C07275=1071.215,48.448,-66.641,172.994,24.716,154.444
C07276=1071.221,48.697,-66.658,172.995,24.719,154.444
C07277=1071.227,48.947,-66.674,172.996,24.722,154.444
C07278=1071.233,49.196,-66.690,172.998,24.724,154.445
C07279=1071.239,49.446,-66.706,172.999,24.727,154.445
C07280=1071.244,49.695,-66.723,173.001,24.730,154.445
C07281=1071.250,49.945,-66.739,173.002,24.733,154.446
C07282=1071.256,50.194,-66.756,173.004,24.735,154.446
C07283=1071.262,50.443,-66.772,173.005,24.738,154.446
C07284=1071.268,50.693,-66.788,173.006,24.741,154.447
C07285=1071.273,50.942,-66.805,173.008,24.743,154.447
C07286=1071.279,51.192,-66.821,173.009,24.746,154.448
C07287=1071.285,51.441,-66.838,173.010,24.748,154.448
C07288=1071.291,51.690,-66.854,173.012,24.751,154.448
C07289=1071.297,51.940,-66.870,173.013,24.754,154.449
C07290=1071.302,52.189,-66.887,173.014,24.757,154.449
C07291=1071.308,52.439,-66.903,173.017,24.759,154.449
C07292=1071.314,52.688,-66.919,173.018,24.762,154.450
C07293=1071.320,52.937,-66.936,173.019,24.764,154.450
C07294=1071.326,53.186,-66.953,173.020,24.767,154.450
C07295=1071.332,53.436,-66.969,173.022,24.770,154.451
C07296=1071.337,53.685,-66.986,173.023,24.773,154.451
C07297=1071.344,53.935,-67.002,173.025,24.775,154.451
C07298=1071.349,54.185,-67.019,173.026,24.778,154.452
C07299=1071.355,54.434,-67.035,173.027,24.780,154.452
C07300=1071.361,54.683,-67.052,173.028,24.783,154.452
C07301=1071.367,54.932,-67.069,173.031,24.786,154.453
C07302=1071.373,55.182,-67.086,173.032,24.789,154.453
C07303=1071.379,55.431,-67.102,173.033,24.791,154.453
C07304=1071.384,55.681,-67.118,173.035,24.794,154.454
C07305=1071.391,55.929,-67.135,173.036,24.796,154.454
C07306=1071.396,56.179,-67.152,173.037,24.799,154.454
C07307=1071.403,56.429,-67.169,173.039,24.802,154.455
C07308=1071.408,56.678,-67.185,173.040,24.805,154.455
C07309=1071.415,56.927,-67.202,173.041,24.807,154.455
C07310=1071.420,57.177,-67.219,173.043,24.810,154.456
C07311=1071.426,57.426,-67.235,173.045,24.812,154.456
C07312=1071.432,57.675,-67.251,173.046,24.815,154.456
C07313=1071.437,57.924,-67.269,173.048,24.818,154.457
C07314=1071.444,58.175,-67.285,173.049,24.821,154.457
C07315=1071.450,58.424,-67.302,173.050,24.823,154.457
C07316=1071.456,58.673,-67.318,173.052,24.826,154.458
C07317=1071.461,58.922,-67.335,173.053,24.828,154.458
C07318=1071.467,59.172,-67.352,173.054,24.831,154.458
C07319=1071.473,59.421,-67.368,173.056,24.833,154.459
C07320=1071.479,59.671,-67.386,173.057,24.836,154.459
C07321=1071.485,59.920,-67.402,173.059,24.839,154.459
C07322=1071.491,60.169,-67.418,173.061,24.841,154.460
C07323=1071.497,60.418,-67.436,173.062,24.844,154.460
C07324=1071.503,60.668,-67.452,173.063,24.847,154.460
C07325=1071.510,60.917,-67.470,173.065,24.850,154.461
C07326=1071.516,61.167,-67.486,173.066,24.852,154.461
C07327=1071.521,61.416,-67.503,173.067,24.855,154.461
C07328=1071.527,61.665,-67.520,173.069,24.857,154.462
C07329=1071.533,61.914,-67.536,173.070,24.860,154.462
C07330=1071.539,62.165,-67.553,173.072,24.863,154.462
C07331=1071.546,62.447,-67.572,173.073,24.866,154.463
C07332=1071.553,62.729,-67.592,173.075,24.869,154.463
C07333=1071.559,63.011,-67.610,173.077,24.872,154.464
C07334=1071.565,63.293,-67.630,173.078,24.875,154.464
C07335=1071.572,63.543,-67.646,173.080,24.877,154.464
C07336=1071.578,63.792,-67.663,173.081,24.879,154.465
C07337=1071.583,64.041,-67.680,173.082,24.882,154.465
C07338=1071.590,64.291,-67.697,173.085,24.885,154.465
C07339=1071.596,64.540,-67.714,173.086,24.888,154.466
C07340=1071.602,64.789,-67.731,173.087,24.890,154.466
C07341=1071.607,65.039,-67.748,173.089,24.893,154.466
C07342=1071.613,65.287,-67.765,173.090,24.895,154.467
C07343=1071.619,65.538,-67.782,173.091,24.898,154.467
C07344=1071.625,65.787,-67.799,173.093,24.901,154.467
C07345=1071.631,66.036,-67.816,173.094,24.904,154.468
C07346=1071.637,66.285,-67.833,173.096,24.906,154.468
C07347=1071.643,66.535,-67.851,173.097,24.909,154.468
C07348=1071.648,66.784,-67.868,173.099,24.911,154.469
C07349=1071.654,67.033,-67.885,173.100,24.914,154.469
C07350=1071.660,67.283,-67.902,173.102,24.917,154.469
C07351=1071.666,67.532,-67.919,173.103,24.920,154.470
C07352=1071.672,67.781,-67.936,173.104,24.922,154.470
C07353=1071.678,68.031,-67.953,173.106,24.925,154.470
C07354=1071.683,68.280,-67.970,173.107,24.927,154.471
C07355=1071.689,68.530,-67.988,173.109,24.930,154.471
C07356=1071.696,68.779,-68.005,173.111,24.933,154.471
C07357=1071.701,69.028,-68.022,173.112,24.936,154.472
C07358=1071.706,69.277,-68.039,173.113,24.939,154.472
C07359=1071.713,69.527,-68.056,173.114,24.941,154.472
C07360=1071.719,69.776,-68.074,173.116,24.944,154.473
C07361=1071.724,70.026,-68.091,173.117,24.946,154.473
C07362=1071.731,70.275,-68.108,173.118,24.949,154.473
C07363=1071.736,70.524,-68.126,173.121,24.952,154.474
C07364=1071.741,70.774,-68.142,173.122,24.955,154.474
C07365=1071.748,71.022,-68.159,173.123,24.957,154.474
C07366=1071.754,71.272,-68.177,173.125,24.960,154.475
C07367=1071.759,71.522,-68.194,173.126,24.962,154.475
C07368=1071.765,71.771,-68.212,173.127,24.965,154.476
C07369=1071.771,72.020,-68.229,173.129,24.967,154.476
C07370=1071.777,72.269,-68.247,173.131,24.971,154.476
C07371=1071.782,72.519,-68.264,173.132,24.973,154.476
C07372=1071.788,72.769,-68.281,173.134,24.976,154.477
C07373=1071.794,73.017,-68.298,173.135,24.979,154.477
C07374=1071.800,73.266,-68.316,173.136,24.981,154.478
C07375=1071.806,73.516,-68.334,173.138,24.984,154.478
C07376=1071.811,73.766,-68.351,173.139,24.986,154.478
C07377=1071.817,74.015,-68.368,173.140,24.989,154.479
C07378=1071.823,74.264,-68.385,173.143,24.992,154.479
C07379=1071.829,74.513,-68.403,173.144,24.995,154.479
C07380=1071.835,74.762,-68.421,173.145,24.997,154.480
C07381=1071.841,75.012,-68.439,173.147,25.000,154.480
C07382=1071.846,75.262,-68.456,173.148,25.002,154.480
C07383=1071.852,75.511,-68.473,173.149,25.005,154.481
C07384=1071.858,75.760,-68.490,173.151,25.008,154.481
C07385=1071.864,76.009,-68.508,173.153,25.011,154.481
C07386=1071.870,76.258,-68.526,173.154,25.013,154.482
C07387=1071.876,76.508,-68.544,173.156,25.016,154.482
C07388=1071.882,76.757,-68.561,173.157,25.018,154.482
C07389=1071.887,77.006,-68.578,173.158,25.021,154.483
C07390=1071.893,77.256,-68.595,173.160,25.024,154.483
C07391=1071.899,77.505,-68.613,173.161,25.026,154.483
C07392=1071.905,77.755,-68.631,173.163,25.029,154.484
C07393=1071.910,78.004,-68.648,173.165,25.032,154.484
C07394=1071.916,78.253,-68.666,173.166,25.034,154.484
C07395=1071.923,78.536,-68.686,173.167,25.037,154.485
C07396=1071.930,78.818,-68.706,173.170,25.040,154.485
C07397=1071.936,79.100,-68.726,173.171,25.043,154.486
C07398=1071.943,79.382,-68.746,173.172,25.046,154.486
C07399=1071.948,79.631,-68.763,173.174,25.049,154.486
C07400=1071.954,79.880,-68.781,173.176,25.052,154.487
C07401=1071.960,80.130,-68.799,173.177,25.055,154.487
C07402=1071.966,80.379,-68.816,173.178,25.058,154.487
C07403=1071.972,80.629,-68.834,173.180,25.060,154.488
C07404=1071.977,80.878,-68.852,173.181,25.063,154.488
C07405=1071.983,81.127,-68.869,173.183,25.065,154.488
C07406=1071.989,81.377,-68.887,173.185,25.068,154.489
C07407=1071.995,81.625,-68.906,173.186,25.071,154.489
C07408=1072.001,81.875,-68.924,173.187,25.074,154.489
C07409=1072.006,82.124,-68.941,173.189,25.076,154.490
C07410=1072.012,82.373,-68.959,173.190,25.079,154.490
C07411=1072.018,82.622,-68.977,173.191,25.082,154.491
C07412=1072.023,82.872,-68.995,173.194,25.084,154.491
C07413=1072.029,83.122,-69.013,173.195,25.087,154.491
C07414=1072.034,83.371,-69.030,173.196,25.090,154.491
C07415=1072.040,83.620,-69.048,173.198,25.092,154.492
C07416=1072.046,83.869,-69.066,173.199,25.095,154.492
C07417=1072.052,84.119,-69.085,173.200,25.098,154.493
C07418=1072.058,84.368,-69.102,173.203,25.100,154.493
C07419=1072.063,84.617,-69.120,173.204,25.103,154.493
C07420=1072.070,84.866,-69.138,173.205,25.105,154.494
C07421=1072.075,85.115,-69.155,173.207,25.108,154.494
C07422=1072.081,85.365,-69.173,173.208,25.111,154.494
C07423=1072.087,85.614,-69.191,173.209,25.114,154.495
C07424=1072.093,85.863,-69.209,173.212,25.116,154.495
C07425=1072.099,86.112,-69.227,173.213,25.119,154.495
C07426=1072.104,86.362,-69.245,173.215,25.121,154.496
C07427=1072.110,86.611,-69.263,173.216,25.124,154.496
C07428=1072.116,86.861,-69.282,173.217,25.127,154.496
C07429=1072.122,87.110,-69.299,173.219,25.130,154.497
C07430=1072.128,87.359,-69.317,173.221,25.132,154.497
C07431=1072.133,87.608,-69.335,173.222,25.135,154.497
C07432=1072.140,87.857,-69.353,173.224,25.137,154.498
C07433=1072.146,88.107,-69.371,173.225,25.140,154.498
C07434=1072.151,88.356,-69.389,173.226,25.143,154.498
C07435=1072.157,88.606,-69.408,173.228,25.146,154.499
C07436=1072.162,88.855,-69.426,173.230,25.148,154.499
C07437=1072.169,89.104,-69.444,173.231,25.150,154.499
C07438=1072.174,89.353,-69.462,173.233,25.153,154.500
C07439=1072.181,89.603,-69.480,173.234,25.156,154.500
C07440=1072.186,89.852,-69.497,173.235,25.159,154.500
C07441=1072.192,90.101,-69.516,173.237,25.161,154.501
C07442=1072.199,90.351,-69.534,173.239,25.164,154.501
C07443=1072.203,90.600,-69.552,173.240,25.166,154.501
C07444=1072.210,90.849,-69.571,173.242,25.169,154.502
C07445=1072.215,91.098,-69.588,173.243,25.172,154.502
C07446=1072.221,91.348,-69.606,173.244,25.175,154.502
C07447=1072.226,91.597,-69.625,173.246,25.177,154.503
C07448=1072.233,91.846,-69.643,173.248,25.180,154.503
C07449=1072.238,92.095,-69.661,173.250,25.182,154.503
C07450=1072.244,92.345,-69.680,173.251,25.185,154.504
C07451=1072.250,92.595,-69.698,173.252,25.188,154.504
C07452=1072.255,92.843,-69.717,173.254,25.190,154.504
C07453=1072.261,93.093,-69.735,173.256,25.193,154.505
C07454=1072.267,93.341,-69.753,173.257,25.196,154.505
C07455=1072.272,93.591,-69.771,173.259,25.198,154.505
C07456=1072.278,93.840,-69.790,173.260,25.201,154.506
C07457=1072.284,94.090,-69.808,173.261,25.204,154.506
C07458=1072.290,94.339,-69.827,173.264,25.207,154.506
C07459=1072.297,94.621,-69.847,173.265,25.210,154.507
C07460=1072.303,94.903,-69.868,173.266,25.212,154.507
C07461=1072.309,95.186,-69.889,173.268,25.216,154.508
C07462=1072.316,95.467,-69.909,173.270,25.219,154.508
C07463=1072.322,95.717,-69.929,173.272,25.221,154.508
C07464=1072.327,95.966,-69.946,173.273,25.224,154.509
C07465=1072.334,96.215,-69.965,173.275,25.226,154.509
C07466=1072.339,96.464,-69.983,173.276,25.229,154.509
C07467=1072.345,96.713,-70.002,173.277,25.232,154.510
C07468=1072.350,96.964,-70.020,173.280,25.235,154.510
C07469=1072.356,97.212,-70.038,173.281,25.237,154.510
C07470=1072.363,97.461,-70.057,173.282,25.240,154.511
C07471=1072.368,97.711,-70.076,173.284,25.242,154.511
C07472=1072.374,97.960,-70.094,173.285,25.245,154.511
C07473=1072.379,98.210,-70.112,173.288,25.248,154.512
C07474=1072.386,98.459,-70.131,173.289,25.251,154.512
C07475=1072.391,98.707,-70.150,173.290,25.253,154.512
C07476=1072.397,98.957,-70.168,173.292,25.255,154.513
C07477=1072.403,99.206,-70.186,173.293,25.258,154.513
C07478=1072.408,99.455,-70.205,173.295,25.261,154.513
C07479=1072.414,99.705,-70.223,173.297,25.264,154.514
C07480=1072.420,99.954,-70.243,173.298,25.266,154.514
C07481=1072.427,100.203,-70.261,173.299,25.269,154.514
C07482=1072.431,100.453,-70.279,173.301,25.271,154.515
C07483=1072.438,100.702,-70.298,173.303,25.274,154.515
C07484=1072.444,100.951,-70.317,173.304,25.277,154.515
C07485=1072.449,101.200,-70.336,173.306,25.279,154.516
C07486=1072.455,101.450,-70.354,173.307,25.282,154.516
C07487=1072.461,101.699,-70.373,173.310,25.285,154.516
C07488=1072.466,101.948,-70.392,173.311,25.287,154.517
C07489=1072.473,102.197,-70.410,173.312,25.290,154.517
C07490=1072.478,102.447,-70.429,173.314,25.293,154.517
C07491=1072.483,102.695,-70.448,173.315,25.295,154.518
C07492=1072.489,102.945,-70.466,173.317,25.298,154.518
C07493=1072.495,103.194,-70.486,173.319,25.300,154.518
C07494=1072.500,103.443,-70.504,173.320,25.303,154.519
C07495=1072.506,103.693,-70.522,173.321,25.306,154.519
C07496=1072.512,103.942,-70.542,173.323,25.309,154.519
C07497=1072.518,104.191,-70.561,173.325,25.311,154.520
C07498=1072.524,104.440,-70.579,173.326,25.314,154.520
C07499=1072.529,104.689,-70.598,173.328,25.316,154.520
C07500=1072.535,104.939,-70.618,173.329,25.319,154.521
C07501=1072.541,105.187,-70.636,173.332,25.322,154.521
C07502=1072.546,105.437,-70.654,173.333,25.325,154.522
C07503=1072.552,105.687,-70.674,173.334,25.327,154.522
C07504=1072.558,105.936,-70.692,173.336,25.330,154.522
C07505=1072.563,106.184,-70.711,173.338,25.333,154.522
C07506=1072.569,106.434,-70.730,173.339,25.335,154.523
C07507=1072.575,106.683,-70.749,173.341,25.338,154.523
C07508=1072.581,106.932,-70.768,173.342,25.341,154.524
C07509=1072.586,107.181,-70.787,173.343,25.343,154.524
C07510=1072.593,107.430,-70.806,173.346,25.346,154.524
C07511=1072.598,107.680,-70.825,173.347,25.348,154.525
C07512=1072.604,107.929,-70.844,173.349,25.351,154.525
C07513=1072.610,108.178,-70.863,173.350,25.354,154.525
C07514=1072.616,108.427,-70.882,173.352,25.356,154.525
C07515=1072.621,108.676,-70.901,173.354,25.359,154.526
C07516=1072.627,108.926,-70.920,173.355,25.361,154.526
C07517=1072.633,109.175,-70.939,173.356,25.364,154.527
C07518=1072.639,109.424,-70.958,173.359,25.367,154.527
C07519=1072.644,109.673,-70.977,173.360,25.369,154.527
C07520=1072.651,109.922,-70.996,173.361,25.372,154.528
C07521=1072.656,110.172,-71.015,173.363,25.374,154.528
C07522=1072.662,110.421,-71.034,173.365,25.378,154.528
C07523=1072.669,110.704,-71.056,173.367,25.380,154.528
C07524=1072.675,110.985,-71.077,173.369,25.383,154.529
C07525=1072.682,111.268,-71.099,173.370,25.386,154.529
C07526=1072.688,111.550,-71.120,173.372,25.389,154.530
C07527=1072.694,111.800,-71.139,173.374,25.391,154.530
C07528=1072.700,112.049,-71.159,173.375,25.394,154.530
C07529=1072.705,112.297,-71.178,173.377,25.397,154.531
C07530=1072.711,112.547,-71.197,173.379,25.400,154.531
C07531=1072.717,112.796,-71.217,173.380,25.402,154.531
C07532=1072.722,113.046,-71.236,173.382,25.405,154.532
C07533=1072.729,113.295,-71.254,173.384,25.408,154.532
C07534=1072.734,113.544,-71.274,173.385,25.410,154.532
C07535=1072.740,113.793,-71.294,173.387,25.413,154.533
C07536=1072.745,114.042,-71.313,173.388,25.415,154.533
C07537=1072.751,114.291,-71.332,173.390,25.418,154.533
C07538=1072.757,114.541,-71.351,173.392,25.421,154.534
C07539=1072.763,114.790,-71.370,173.393,25.423,154.534
C07540=1072.768,115.039,-71.390,173.395,25.426,154.534
C07541=1072.774,115.288,-71.410,173.397,25.429,154.535
C07542=1072.779,115.537,-71.428,173.398,25.431,154.535
C07543=1072.785,115.786,-71.448,173.400,25.434,154.535
C07544=1072.791,116.035,-71.468,173.401,25.437,154.536
C07545=1072.797,116.285,-71.487,173.403,25.440,154.536
C07546=1072.802,116.534,-71.506,173.405,25.442,154.536
C07547=1072.807,116.784,-71.526,173.406,25.445,154.537
C07548=1072.813,117.032,-71.546,173.408,25.448,154.537
C07549=1072.818,117.281,-71.565,173.410,25.450,154.537
C07550=1072.824,117.531,-71.584,173.411,25.453,154.538
C07551=1072.830,117.780,-71.604,173.412,25.455,154.538
C07552=1072.836,118.029,-71.623,173.415,25.458,154.538
C07553=1072.841,118.278,-71.642,173.416,25.461,154.539
C07554=1072.847,118.527,-71.662,173.418,25.463,154.539
C07555=1072.853,118.777,-71.682,173.419,25.466,154.539
C07556=1072.858,119.025,-71.701,173.421,25.469,154.540
C07557=1072.863,119.275,-71.721,173.423,25.471,154.540
C07558=1072.869,119.524,-71.740,173.424,25.474,154.540
C07559=1072.875,119.773,-71.760,173.426,25.477,154.541
C07560=1072.881,120.022,-71.780,173.428,25.479,154.541
C07561=1072.886,120.272,-71.799,173.429,25.482,154.541
C07562=1072.892,120.520,-71.819,173.431,25.484,154.542
C07563=1072.898,120.770,-71.838,173.433,25.488,154.542
C07564=1072.904,121.019,-71.858,173.434,25.490,154.542
C07565=1072.909,121.268,-71.878,173.436,25.492,154.543
C07566=1072.915,121.518,-71.897,173.438,25.495,154.543
C07567=1072.921,121.767,-71.917,173.439,25.498,154.543
C07568=1072.926,122.016,-71.936,173.441,25.501,154.544
C07569=1072.932,122.265,-71.956,173.443,25.503,154.544
C07570=1072.938,122.514,-71.975,173.444,25.506,154.544
C07571=1072.944,122.763,-71.995,173.446,25.508,154.545
C07572=1072.949,123.013,-72.015,173.447,25.511,154.545
C07573=1072.955,123.262,-72.035,173.450,25.514,154.545
C07574=1072.961,123.511,-72.054,173.451,25.516,154.546
C07575=1072.967,123.760,-72.074,173.452,25.519,154.546
C07576=1072.972,124.009,-72.094,173.455,25.522,154.546
C07577=1072.978,124.258,-72.114,173.456,25.524,154.547
C07578=1072.984,124.507,-72.134,173.458,25.527,154.547
C07579=1072.989,124.757,-72.153,173.460,25.529,154.547
C07580=1072.995,125.006,-72.173,173.461,25.532,154.548
C07581=1073.001,125.255,-72.193,173.463,25.535,154.548
C07582=1073.007,125.504,-72.213,173.465,25.537,154.548
C07583=1073.012,125.754,-72.232,173.466,25.540,154.549
C07584=1073.018,126.002,-72.252,173.468,25.542,154.549
C07585=1073.024,126.251,-72.272,173.469,25.545,154.549
C07586=1073.030,126.501,-72.292,173.472,25.548,154.550
C07587=1073.036,126.783,-72.314,173.473,25.551,154.550
C07588=1073.043,127.065,-72.336,173.475,25.553,154.550
C07589=1073.049,127.347,-72.359,173.478,25.556,154.551
C07590=1073.055,127.630,-72.382,173.479,25.559,154.551
C07591=1073.061,127.878,-72.402,173.481,25.562,154.551
C07592=1073.067,128.127,-72.422,173.483,25.565,154.552
C07593=1073.073,128.376,-72.442,173.484,25.567,154.552
C07594=1073.078,128.626,-72.461,173.486,25.570,154.552
C07595=1073.084,128.875,-72.481,173.488,25.572,154.553
C07596=1073.090,129.123,-72.501,173.489,25.575,154.553
C07597=1073.097,129.374,-72.521,173.492,25.577,154.553
C07598=1073.102,129.623,-72.541,173.493,25.580,154.554
C07599=1073.108,129.871,-72.561,173.494,25.583,154.554
C07600=1073.114,130.120,-72.581,173.497,25.585,154.554
C07601=1073.120,130.370,-72.601,173.498,25.588,154.555
C07602=1073.125,130.619,-72.621,173.500,25.590,154.555
C07603=1073.131,130.868,-72.641,173.502,25.593,154.555
C07604=1073.137,131.117,-72.661,173.503,25.595,154.555
C07605=1073.143,131.366,-72.681,173.505,25.598,154.556
C07606=1073.148,131.616,-72.701,173.507,25.601,154.556
C07607=1073.154,131.865,-72.721,173.509,25.603,154.556
C07608=1073.160,132.113,-72.741,173.510,25.606,154.557
C07609=1073.166,132.362,-72.762,173.512,25.608,154.557
C07610=1073.172,132.611,-72.782,173.514,25.611,154.557
C07611=1073.177,132.860,-72.802,173.515,25.614,154.558
C07612=1073.183,133.111,-72.822,173.517,25.616,154.558
C07613=1073.188,133.360,-72.842,173.519,25.619,154.558
C07614=1073.194,133.608,-72.862,173.521,25.622,154.559
C07615=1073.200,133.858,-72.883,173.523,25.625,154.559
C07616=1073.206,134.106,-72.903,173.524,25.627,154.559
C07617=1073.211,134.356,-72.923,173.526,25.629,154.560
C07618=1073.217,134.604,-72.943,173.528,25.632,154.560
C07619=1073.223,134.854,-72.964,173.529,25.635,154.560
C07620=1073.229,135.103,-72.984,173.532,25.637,154.561
C07621=1073.234,135.352,-73.005,173.533,25.640,154.561
C07622=1073.240,135.601,-73.025,173.534,25.642,154.561
C07623=1073.245,135.850,-73.045,173.537,25.645,154.562
C07624=1073.251,136.099,-73.065,173.538,25.648,154.562
C07625=1073.257,136.349,-73.086,173.540,25.650,154.562
C07626=1073.263,136.597,-73.106,173.542,25.653,154.563
C07627=1073.268,136.847,-73.127,173.543,25.655,154.563
C07628=1073.274,137.095,-73.147,173.546,25.658,154.563
C07629=1073.280,137.345,-73.167,173.547,25.661,154.564
C07630=1073.286,137.593,-73.187,173.548,25.663,154.564
C07631=1073.292,137.843,-73.208,173.551,25.666,154.564
C07632=1073.297,138.092,-73.229,173.552,25.669,154.564
C07633=1073.303,138.341,-73.249,173.555,25.671,154.565
C07634=1073.308,138.590,-73.269,173.556,25.674,154.565
C07635=1073.315,138.840,-73.289,173.557,25.676,154.565
C07636=1073.320,139.089,-73.310,173.560,25.679,154.566
C07637=1073.325,139.338,-73.331,173.561,25.682,154.566
C07638=1073.331,139.587,-73.351,173.563,25.684,154.566
C07639=1073.337,139.835,-73.372,173.565,25.687,154.567
C07640=1073.343,140.085,-73.392,173.566,25.690,154.567
C07641=1073.349,140.334,-73.413,173.569,25.692,154.567
C07642=1073.354,140.583,-73.433,173.570,25.695,154.568
C07643=1073.360,140.832,-73.453,173.572,25.697,154.568
C07644=1073.366,141.082,-73.474,173.574,25.700,154.568
C07645=1073.371,141.330,-73.495,173.575,25.703,154.569
C07646=1073.376,141.579,-73.516,173.578,25.705,154.569
C07647=1073.382,141.828,-73.536,173.579,25.708,154.569
C07648=1073.388,142.078,-73.557,173.580,25.711,154.570
C07649=1073.394,142.327,-73.577,173.583,25.713,154.570
C07650=1073.399,142.576,-73.599,173.584,25.715,154.570
C07651=1073.405,142.858,-73.621,173.587,25.719,154.571
C07652=1073.412,143.140,-73.645,173.589,25.722,154.571
C07653=1073.419,143.422,-73.668,173.590,25.725,154.571
C07654=1073.425,143.704,-73.692,173.592,25.728,154.572
C07655=1073.431,143.953,-73.712,173.595,25.730,154.572
C07656=1073.436,144.202,-73.733,173.596,25.733,154.572
C07657=1073.442,144.451,-73.755,173.598,25.735,154.573
C07658=1073.448,144.700,-73.775,173.600,25.738,154.573
C07659=1073.453,144.949,-73.796,173.602,25.740,154.573
C07660=1073.460,145.198,-73.817,173.604,25.743,154.574
C07661=1073.465,145.447,-73.837,173.605,25.746,154.574
C07662=1073.470,145.697,-73.858,173.608,25.748,154.574
C07663=1073.476,145.945,-73.879,173.609,25.751,154.575
C07664=1073.482,146.195,-73.900,173.611,25.753,154.575
C07665=1073.488,146.444,-73.920,173.613,25.756,154.575
C07666=1073.493,146.692,-73.941,173.614,25.759,154.576
C07667=1073.499,146.942,-73.962,173.617,25.762,154.576
C07668=1073.505,147.191,-73.983,173.618,25.764,154.576
C07669=1073.511,147.440,-74.004,173.620,25.767,154.576
C07670=1073.517,147.689,-74.024,173.622,25.769,154.577
C07671=1073.522,147.938,-74.046,173.623,25.772,154.577
C07672=1073.528,148.188,-74.067,173.626,25.775,154.577
C07673=1073.533,148.436,-74.088,173.627,25.777,154.578
C07674=1073.539,148.685,-74.108,173.630,25.780,154.578
C07675=1073.545,148.934,-74.130,173.631,25.782,154.578
C07676=1073.550,149.183,-74.151,173.633,25.785,154.579
C07677=1073.556,149.432,-74.172,173.635,25.788,154.579
C07678=1073.562,149.682,-74.193,173.637,25.790,154.579
C07679=1073.567,149.930,-74.214,173.638,25.793,154.580
C07680=1073.572,150.179,-74.235,173.640,25.796,154.580
C07681=1073.579,150.429,-74.256,173.642,25.798,154.580
C07682=1073.584,150.678,-74.277,173.644,25.800,154.581
C07683=1073.590,150.927,-74.298,173.646,25.804,154.581
C07684=1073.595,151.176,-74.319,173.647,25.806,154.581
C07685=1073.601,151.425,-74.340,173.650,25.808,154.581
C07686=1073.607,151.674,-74.362,173.651,25.811,154.582
C07687=1073.612,151.923,-74.382,173.654,25.814,154.582
C07688=1073.618,152.172,-74.404,173.655,25.817,154.583
C07689=1073.624,152.421,-74.425,173.657,25.819,154.583
C07690=1073.629,152.670,-74.446,173.659,25.822,154.583
C07691=1073.635,152.919,-74.467,173.660,25.824,154.584
C07692=1073.641,153.168,-74.488,173.663,25.827,154.584
C07693=1073.647,153.417,-74.510,173.664,25.829,154.584
C07694=1073.652,153.666,-74.531,173.666,25.832,154.584
C07695=1073.658,153.915,-74.551,173.668,25.835,154.585
C07696=1073.664,154.164,-74.573,173.670,25.837,154.585
C07697=1073.669,154.413,-74.594,173.672,25.840,154.585
C07698=1073.675,154.662,-74.615,173.674,25.843,154.586
C07699=1073.681,154.911,-74.637,173.676,25.845,154.586
C07700=1073.687,155.160,-74.658,173.678,25.848,154.586
C07701=1073.691,155.410,-74.679,173.679,25.850,154.587
C07702=1073.698,155.659,-74.701,173.682,25.853,154.587
C07703=1073.703,155.907,-74.722,173.683,25.856,154.587
C07704=1073.709,156.156,-74.744,173.685,25.858,154.588
C07705=1073.715,156.406,-74.764,173.687,25.861,154.588
C07706=1073.720,156.654,-74.786,173.689,25.864,154.588
C07707=1073.726,156.904,-74.808,173.691,25.866,154.588
C07708=1073.731,157.152,-74.829,173.693,25.869,154.589
C07709=1073.737,157.401,-74.851,173.694,25.872,154.589
C07710=1073.743,157.650,-74.871,173.697,25.874,154.589
C07711=1073.749,157.900,-74.893,173.698,25.877,154.590
C07712=1073.754,158.148,-74.914,173.701,25.880,154.590
C07713=1073.760,158.398,-74.937,173.702,25.882,154.590
C07714=1073.765,158.646,-74.958,173.704,25.885,154.591
C07715=1073.772,158.929,-74.982,173.707,25.888,154.591
C07716=1073.779,159.210,-75.006,173.708,25.890,154.591
C07717=1073.784,159.492,-75.030,173.710,25.893,154.592
C07718=1073.791,159.774,-75.055,173.713,25.897,154.592
C07719=1073.797,160.023,-75.077,173.715,25.899,154.592
C07720=1073.803,160.272,-75.098,173.717,25.901,154.593
C07721=1073.808,160.520,-75.120,173.719,25.905,154.593
C07722=1073.814,160.770,-75.142,173.720,25.907,154.593
C07723=1073.819,161.018,-75.163,173.723,25.909,154.594
C07724=1073.826,161.267,-75.185,173.724,25.912,154.594
C07725=1073.832,161.517,-75.206,173.727,25.915,154.594
C07726=1073.837,161.766,-75.228,173.728,25.918,154.595
C07727=1073.841,162.014,-75.250,173.730,25.920,154.595
C07728=1073.848,162.264,-75.272,173.732,25.923,154.595
C07729=1073.852,162.512,-75.294,173.734,25.926,154.596
C07730=1073.858,162.762,-75.315,173.736,25.928,154.596
C07731=1073.866,163.133,-75.347,173.739,25.933,154.597
C07732=1073.874,163.505,-75.381,173.742,25.937,154.597
C07733=1073.883,163.877,-75.412,173.745,25.941,154.597
C07734=1073.891,164.249,-75.445,173.747,25.944,154.598
C07735=1073.896,164.498,-75.467,173.749,25.947,154.598
C07736=1073.902,164.747,-75.489,173.752,25.950,154.599
C07737=1073.907,164.996,-75.511,173.753,25.953,154.599
C07738=1073.913,165.245,-75.532,173.755,25.955,154.599
C07739=1073.918,165.494,-75.554,173.757,25.958,154.600
C07740=1073.924,165.742,-75.577,173.759,25.961,154.600
C07741=1073.930,165.992,-75.599,173.761,25.963,154.600
C07742=1073.935,166.240,-75.620,173.763,25.966,154.601
C07743=1073.941,166.490,-75.642,173.764,25.968,154.601
C07744=1073.946,166.739,-75.664,173.767,25.972,154.601
C07745=1073.952,166.987,-75.687,173.769,25.974,154.602
C07746=1073.957,167.236,-75.708,173.771,25.977,154.602
C07747=1073.963,167.485,-75.730,173.773,25.979,154.602
C07748=1073.969,167.735,-75.752,173.774,25.982,154.603
C07749=1073.973,167.984,-75.774,173.777,25.985,154.603
C07750=1073.980,168.232,-75.797,173.778,25.987,154.603
C07751=1073.985,168.481,-75.818,173.781,25.990,154.604
C07752=1073.991,168.730,-75.840,173.782,25.993,154.604
C07753=1073.996,168.980,-75.862,173.784,25.996,154.604
C07754=1074.001,169.228,-75.885,173.787,25.998,154.605
C07755=1074.008,169.477,-75.907,173.788,26.001,154.605
C07756=1074.013,169.727,-75.929,173.791,26.004,154.605
C07757=1074.019,169.975,-75.951,173.792,26.006,154.606
C07758=1074.024,170.224,-75.973,173.794,26.009,154.606
C07759=1074.030,170.474,-75.995,173.797,26.012,154.606
C07760=1074.036,170.721,-76.017,173.798,26.014,154.607
C07761=1074.041,170.971,-76.039,173.801,26.017,154.607
C07762=1074.046,171.221,-76.062,173.802,26.019,154.607
C07763=1074.052,171.468,-76.084,173.804,26.022,154.608
C07764=1074.058,171.718,-76.106,173.807,26.025,154.608
C07765=1074.063,171.967,-76.129,173.808,26.027,154.608
C07766=1074.069,172.215,-76.150,173.811,26.030,154.608
C07767=1074.074,172.465,-76.172,173.812,26.033,154.609
C07768=1074.080,172.714,-76.195,173.814,26.036,154.609
C07769=1074.086,172.963,-76.217,173.817,26.038,154.609
C07770=1074.091,173.211,-76.239,173.818,26.041,154.610
C07771=1074.097,173.461,-76.262,173.821,26.044,154.610
C07772=1074.103,173.709,-76.284,173.822,26.046,154.610
C07773=1074.109,173.959,-76.306,173.824,26.049,154.611
C07774=1074.114,174.207,-76.329,173.827,26.052,154.611
C07775=1074.123,174.614,-76.365,173.830,26.056,154.611
C07776=1074.132,175.022,-76.401,173.833,26.060,154.612
C07777=1074.142,175.430,-76.437,173.837,26.064,154.612
C07778=1074.152,175.838,-76.475,173.840,26.069,154.613
C07779=1074.156,176.087,-76.497,173.841,26.071,154.613
C07780=1074.163,176.335,-76.519,173.844,26.074,154.614
C07781=1074.169,176.584,-76.542,173.846,26.077,154.614
C07782=1074.174,176.834,-76.565,173.848,26.079,154.614
C07783=1074.180,177.082,-76.587,173.850,26.082,154.615
C07784=1074.185,177.331,-76.609,173.852,26.085,154.615
C07785=1074.191,177.580,-76.632,173.854,26.087,154.615
C07786=1074.197,177.829,-76.655,173.856,26.090,154.616
C07787=1074.203,178.078,-76.676,173.859,26.093,154.616
C07788=1074.209,178.327,-76.699,173.860,26.095,154.616
C07789=1074.215,178.576,-76.722,173.863,26.098,154.616
C07790=1074.220,178.825,-76.744,173.865,26.101,154.617
C07791=1074.226,179.073,-76.766,173.866,26.103,154.617
C07792=1074.232,179.322,-76.789,173.869,26.106,154.617
C07793=1074.237,179.572,-76.812,173.871,26.109,154.618
C07794=1074.243,179.820,-76.835,173.873,26.111,154.618
C07795=1074.249,180.069,-76.857,173.875,26.114,154.618
C07796=1074.255,180.318,-76.880,173.877,26.117,154.619
C07797=1074.260,180.567,-76.902,173.879,26.119,154.619
C07798=1074.266,180.816,-76.925,173.881,26.121,154.619
C07799=1074.272,181.065,-76.948,173.884,26.125,154.620
C07800=1074.278,181.313,-76.970,173.885,26.127,154.620
C07801=1074.283,181.563,-76.992,173.887,26.129,154.620
C07802=1074.289,181.812,-77.015,173.890,26.132,154.620
C07803=1074.295,182.060,-77.038,173.891,26.135,154.621
C07804=1074.300,182.309,-77.061,173.894,26.137,154.621
C07805=1074.307,182.558,-77.083,173.896,26.140,154.621
C07806=1074.312,182.807,-77.106,173.898,26.143,154.622
C07807=1074.318,183.056,-77.129,173.900,26.145,154.622
C07808=1074.324,183.305,-77.151,173.902,26.148,154.622
C07809=1074.329,183.554,-77.174,173.904,26.150,154.623
C07810=1074.336,183.803,-77.197,173.906,26.153,154.623
C07811=1074.342,184.052,-77.220,173.909,26.156,154.623
C07812=1074.347,184.301,-77.243,173.911,26.158,154.624
C07813=1074.353,184.549,-77.266,173.912,26.161,154.624
C07814=1074.359,184.798,-77.289,173.915,26.164,154.624
C07815=1074.364,185.047,-77.311,173.917,26.166,154.624
C07816=1074.370,185.296,-77.334,173.919,26.169,154.625
C07817=1074.376,185.545,-77.357,173.921,26.172,154.625
C07818=1074.381,185.793,-77.380,173.923,26.175,154.626
C07819=1074.386,186.042,-77.404,173.925,26.177,154.626
C07820=1074.392,186.291,-77.426,173.927,26.180,154.626
C07821=1074.398,186.540,-77.449,173.930,26.183,154.627
C07822=1074.403,186.789,-77.472,173.932,26.186,154.627
C07823=1074.408,187.038,-77.496,173.933,26.189,154.627
C07824=1074.414,187.287,-77.519,173.936,26.191,154.628
C07825=1074.420,187.536,-77.542,173.938,26.194,154.628
C07826=1074.425,187.785,-77.565,173.940,26.196,154.628
C07827=1074.430,188.034,-77.588,173.942,26.200,154.629
C07828=1074.436,188.283,-77.611,173.944,26.202,154.629
C07829=1074.441,188.531,-77.634,173.947,26.205,154.629
C07830=1074.447,188.780,-77.657,173.948,26.208,154.630
C07831=1074.452,189.029,-77.680,173.951,26.211,154.630
C07832=1074.458,189.278,-77.704,173.953,26.213,154.630
C07833=1074.464,189.527,-77.727,173.955,26.216,154.631
C07834=1074.469,189.775,-77.750,173.957,26.219,154.631
C07835=1074.474,190.025,-77.773,173.959,26.222,154.631
C07836=1074.480,190.274,-77.796,173.962,26.224,154.632
C07837=1074.486,190.522,-77.819,173.964,26.227,154.632
C07838=1074.491,190.771,-77.844,173.965,26.230,154.632
C07839=1074.498,191.052,-77.869,173.968,26.233,154.633
C07840=1074.504,191.334,-77.895,173.970,26.236,154.633
C07841=1074.511,191.615,-77.922,173.973,26.239,154.633
C07842=1074.517,191.895,-77.948,173.976,26.242,154.634
C07843=1074.522,192.144,-77.972,173.977,26.245,154.634
C07844=1074.528,192.393,-77.995,173.979,26.248,154.634
C07845=1074.534,192.642,-78.018,173.982,26.251,154.635
C07846=1074.539,192.891,-78.041,173.984,26.253,154.635
C07847=1074.545,193.139,-78.065,173.987,26.256,154.635
C07848=1074.551,193.388,-78.088,173.988,26.259,154.636
C07849=1074.556,193.637,-78.112,173.990,26.262,154.636
C07850=1074.562,193.886,-78.135,173.993,26.264,154.636
C07851=1074.567,194.135,-78.158,173.995,26.267,154.637
C07852=1074.573,194.385,-78.182,173.997,26.270,154.637
C07853=1074.579,194.633,-78.206,173.999,26.273,154.637
C07854=1074.585,194.882,-78.229,174.001,26.275,154.638
C07855=1074.590,195.130,-78.253,174.004,26.278,154.638
C07856=1074.596,195.379,-78.276,174.006,26.281,154.638
C07857=1074.601,195.628,-78.299,174.008,26.284,154.639
C07858=1074.607,195.877,-78.323,174.010,26.286,154.639
C07859=1074.612,196.126,-78.346,174.012,26.289,154.639
C07860=1074.619,196.374,-78.370,174.015,26.292,154.640
C07861=1074.624,196.624,-78.394,174.017,26.295,154.640
C07862=1074.630,196.872,-78.417,174.019,26.297,154.640
C07863=1074.635,197.121,-78.441,174.021,26.300,154.641
C07864=1074.641,197.369,-78.465,174.023,26.303,154.641
C07865=1074.647,197.618,-78.487,174.026,26.305,154.641
C07866=1074.652,197.867,-78.512,174.028,26.308,154.642
C07867=1074.659,198.117,-78.535,174.030,26.311,154.642
C07868=1074.664,198.365,-78.559,174.032,26.314,154.642
C07869=1074.670,198.614,-78.582,174.034,26.316,154.643
C07870=1074.676,198.862,-78.606,174.037,26.319,154.643
C07871=1074.681,199.112,-78.629,174.039,26.322,154.643
C07872=1074.687,199.360,-78.653,174.042,26.325,154.644
C07873=1074.692,199.610,-78.677,174.043,26.327,154.644
C07874=1074.698,199.858,-78.701,174.045,26.330,154.644
C07875=1074.704,200.106,-78.724,174.048,26.333,154.645
C07876=1074.709,200.355,-78.748,174.050,26.336,154.645
C07877=1074.716,200.604,-78.772,174.053,26.339,154.645
C07878=1074.721,200.853,-78.796,174.055,26.342,154.646
C07879=1074.727,201.102,-78.819,174.056,26.344,154.646
C07880=1074.732,201.351,-78.843,174.059,26.346,154.646
C07881=1074.739,201.600,-78.867,174.061,26.350,154.647
C07882=1074.745,201.848,-78.890,174.064,26.352,154.647
C07883=1074.750,202.097,-78.915,174.066,26.355,154.647
C07884=1074.756,202.345,-78.938,174.068,26.358,154.647
C07885=1074.762,202.595,-78.962,174.070,26.361,154.648
C07886=1074.767,202.844,-78.986,174.072,26.363,154.648
C07887=1074.773,203.092,-79.010,174.075,26.366,154.649
C07888=1074.778,203.341,-79.034,174.077,26.369,154.649
C07889=1074.784,203.591,-79.058,174.079,26.372,154.649
C07890=1074.790,203.839,-79.082,174.082,26.375,154.650
C07891=1074.795,204.087,-79.106,174.084,26.378,154.650
C07892=1074.800,204.336,-79.130,174.086,26.380,154.650
C07893=1074.807,204.585,-79.154,174.088,26.383,154.651
C07894=1074.812,204.834,-79.179,174.090,26.386,154.651
C07895=1074.817,205.083,-79.202,174.093,26.389,154.651
C07896=1074.823,205.331,-79.227,174.095,26.392,154.652
C07897=1074.829,205.580,-79.251,174.098,26.395,154.652
C07898=1074.835,205.829,-79.275,174.100,26.398,154.652
C07899=1074.840,206.078,-79.299,174.102,26.400,154.653
C07900=1074.845,206.326,-79.323,174.105,26.403,154.653
C07901=1074.852,206.575,-79.347,174.106,26.406,154.653
C07902=1074.857,206.824,-79.372,174.109,26.409,154.654
C07903=1074.881,207.863,-79.472,174.229,26.472,154.654
C07904=1074.890,208.275,-79.513,174.232,26.478,154.655
C07905=1074.899,208.688,-79.554,174.235,26.484,154.656
C07906=1074.910,209.100,-79.596,174.239,26.491,154.657
C07907=1074.919,209.512,-79.637,174.243,26.497,154.658
C07908=1074.925,209.761,-79.662,174.245,26.501,154.658
C07909=1074.931,210.009,-79.687,174.247,26.504,154.659
C07910=1074.936,210.259,-79.711,174.249,26.509,154.660
C07911=1074.942,210.507,-79.736,174.252,26.512,154.660
C07912=1074.948,210.755,-79.762,174.254,26.516,154.661
C07913=1074.954,211.005,-79.786,174.256,26.520,154.661
C07914=1074.960,211.253,-79.811,174.257,26.523,154.662
C07915=1074.965,211.502,-79.836,174.259,26.527,154.662
C07916=1074.971,211.751,-79.862,174.262,26.531,154.663
C07917=1074.977,211.999,-79.887,174.264,26.534,154.663
C07918=1074.983,212.248,-79.911,174.266,26.539,154.664
C07919=1074.988,212.496,-79.936,174.268,26.542,154.665
C07920=1074.994,212.745,-79.961,174.270,26.546,154.665
C07921=1075.000,212.994,-79.986,174.272,26.550,154.666
C07922=1075.005,213.242,-80.012,174.275,26.554,154.666
C07923=1075.011,213.492,-80.036,174.277,26.557,154.667
C07924=1075.017,213.740,-80.062,174.279,26.561,154.667
C07925=1075.023,213.988,-80.087,174.281,26.565,154.668
C07926=1075.028,214.237,-80.113,174.283,26.569,154.669
C07927=1075.034,214.487,-80.137,174.286,26.573,154.669
C07928=1075.040,214.734,-80.162,174.288,26.576,154.670
C07929=1075.045,214.983,-80.188,174.290,26.580,154.670
C07930=1075.052,215.232,-80.214,174.292,26.584,154.671
C07931=1075.057,215.480,-80.239,174.295,26.587,154.671
C07932=1075.063,215.729,-80.263,174.297,26.592,154.672
C07933=1075.069,215.978,-80.289,174.299,26.595,154.672
C07934=1075.074,216.226,-80.314,174.301,26.599,154.673
C07935=1075.080,216.475,-80.339,174.302,26.603,154.674
C07936=1075.086,216.724,-80.365,174.305,26.606,154.674
C07937=1075.092,216.973,-80.391,174.307,26.610,154.675
C07938=1075.097,217.221,-80.415,174.309,26.614,154.675
C07939=1075.103,217.470,-80.441,174.311,26.618,154.676
C07940=1075.109,217.719,-80.466,174.313,26.622,154.676
C07941=1075.115,217.968,-80.492,174.316,26.625,154.677
C07942=1075.120,218.216,-80.517,174.318,26.629,154.678
C07943=1075.126,218.465,-80.542,174.320,26.633,154.678
C07944=1075.133,218.713,-80.568,174.322,26.637,154.679
C07945=1075.138,218.962,-80.594,174.324,26.640,154.679
C07946=1075.144,219.210,-80.619,174.327,26.644,154.680
C07947=1075.149,219.459,-80.645,174.329,26.648,154.680
C07948=1075.155,219.708,-80.670,174.331,26.651,154.681
C07949=1075.161,219.956,-80.695,174.333,26.655,154.681
C07950=1075.167,220.205,-80.721,174.336,26.659,154.682
C07951=1075.173,220.454,-80.747,174.338,26.663,154.683
C07952=1075.179,220.702,-80.772,174.340,26.666,154.683
C07953=1075.184,220.951,-80.797,174.342,26.670,154.684
C07954=1075.190,221.200,-80.823,174.344,26.674,154.684
C07955=1075.196,221.449,-80.849,174.347,26.678,154.685
C07956=1075.205,221.865,-80.892,174.350,26.684,154.686
C07957=1075.215,222.282,-80.935,174.354,26.690,154.687
C07958=1075.225,222.698,-80.978,174.358,26.697,154.688
C07959=1075.234,223.114,-81.021,174.361,26.703,154.689
C07960=1075.241,223.363,-81.047,174.364,26.706,154.689
C07961=1075.246,223.612,-81.072,174.366,26.711,154.690
C07962=1075.252,223.861,-81.098,174.368,26.714,154.690
C07963=1075.258,224.110,-81.124,174.370,26.718,154.691
C07964=1075.263,224.357,-81.150,174.372,26.722,154.691
C07965=1075.268,224.606,-81.176,174.375,26.725,154.692
C07966=1075.275,224.855,-81.201,174.377,26.729,154.692
C07967=1075.280,225.104,-81.227,174.379,26.733,154.693
C07968=1075.287,225.352,-81.253,174.382,26.737,154.694
C07969=1075.292,225.601,-81.279,174.385,26.741,154.694
C07970=1075.298,225.850,-81.305,174.387,26.745,154.695
C07971=1075.304,226.098,-81.331,174.389,26.748,154.695
C07972=1075.310,226.347,-81.357,174.391,26.752,154.696
C07973=1075.315,226.596,-81.383,174.393,26.756,154.696
C07974=1075.321,226.843,-81.409,174.396,26.760,154.697
C07975=1075.326,227.092,-81.435,174.398,26.763,154.697
C07976=1075.332,227.341,-81.461,174.400,26.767,154.698
C07977=1075.338,227.589,-81.487,174.402,26.771,154.699
C07978=1075.344,227.838,-81.513,174.405,26.774,154.699
C07979=1075.350,228.087,-81.539,174.407,26.778,154.700
C07980=1075.356,228.335,-81.565,174.409,26.782,154.700
C07981=1075.361,228.584,-81.591,174.411,26.786,154.701
C07982=1075.367,228.833,-81.617,174.414,26.789,154.701
C07983=1075.373,229.081,-81.643,174.416,26.793,154.702
C07984=1075.379,229.330,-81.669,174.418,26.797,154.702
C07985=1075.385,229.579,-81.695,174.420,26.800,154.703
C07986=1075.391,229.827,-81.721,174.423,26.804,154.704
C07987=1075.397,230.076,-81.747,174.425,26.808,154.704
C07988=1075.402,230.324,-81.774,174.427,26.812,154.705
C07989=1075.408,230.573,-81.800,174.429,26.815,154.705
C07990=1075.414,230.822,-81.826,174.432,26.819,154.706
C07991=1075.419,231.070,-81.853,174.435,26.823,154.706
C07992=1075.426,231.319,-81.878,174.437,26.827,154.707
C07993=1075.431,231.567,-81.905,174.439,26.830,154.707
C07994=1075.437,231.816,-81.931,174.441,26.834,154.708
C07995=1075.443,232.064,-81.958,174.444,26.838,154.709
C07996=1075.448,232.313,-81.984,174.446,26.842,154.709
C07997=1075.454,232.562,-82.010,174.448,26.846,154.710
C07998=1075.460,232.810,-82.037,174.450,26.849,154.710
C07999=1075.465,233.058,-82.063,174.453,26.853,154.711
C08000=1075.471,233.307,-82.089,174.455,26.857,154.711
C08001=1075.477,233.555,-82.115,174.457,26.860,154.712
C08002=1075.483,233.804,-82.142,174.459,26.864,154.712
C08003=1075.489,234.052,-82.169,174.462,26.868,154.713
C08004=1075.494,234.301,-82.195,174.465,26.872,154.714
C08005=1075.501,234.550,-82.222,174.467,26.875,154.714
C08006=1075.506,234.798,-82.248,174.469,26.880,154.715
C08007=1075.512,235.047,-82.275,174.471,26.883,154.715
C08008=1075.519,235.390,-82.312,174.474,26.888,154.716
C08009=1075.528,235.734,-82.348,174.477,26.894,154.717
C08010=1075.535,236.077,-82.385,174.481,26.899,154.718
C08011=1075.543,236.420,-82.422,174.484,26.904,154.718
C08012=1075.549,236.669,-82.448,174.486,26.908,154.719
C08013=1075.555,236.917,-82.474,174.489,26.911,154.719
C08014=1075.560,237.166,-82.501,174.491,26.915,154.720
C08015=1075.567,237.415,-82.528,174.493,26.919,154.721
C08016=1075.573,237.663,-82.555,174.496,26.923,154.721
C08017=1075.578,237.912,-82.581,174.499,26.926,154.722
C08018=1075.584,238.160,-82.608,174.501,26.930,154.722
C08019=1075.590,238.408,-82.635,174.503,26.934,154.723
C08020=1075.595,238.657,-82.662,174.505,26.938,154.723
C08021=1075.601,238.906,-82.689,174.508,26.942,154.724
C08022=1075.607,239.154,-82.716,174.510,26.945,154.724
C08023=1075.613,239.403,-82.742,174.512,26.949,154.725
C08024=1075.621,239.716,-82.776,174.515,26.954,154.726
C08025=1075.628,240.030,-82.809,174.518,26.958,154.726
C08026=1075.634,240.343,-82.843,174.521,26.963,154.727
C08027=1075.642,240.656,-82.877,174.524,26.968,154.728
C08028=1075.648,240.905,-82.905,174.527,26.971,154.728
C08029=1075.654,241.154,-82.931,174.529,26.975,154.729
C08030=1075.659,241.402,-82.958,174.532,26.979,154.729
C08031=1075.665,241.650,-82.984,174.534,26.983,154.730
C08032=1075.672,241.899,-83.012,174.537,26.986,154.731
C08033=1075.678,242.147,-83.039,174.539,26.991,154.731
C08034=1075.683,242.396,-83.066,174.541,26.994,154.732
C08035=1075.689,242.644,-83.093,174.543,26.998,154.732
C08036=1075.695,242.893,-83.120,174.546,27.001,154.733
C08037=1075.701,243.142,-83.146,174.549,27.006,154.733
C08038=1075.706,243.390,-83.174,174.551,27.009,154.734
C08039=1075.712,243.638,-83.201,174.553,27.013,154.734
C08040=1075.718,243.886,-83.228,174.556,27.017,154.735
C08041=1075.723,244.136,-83.255,174.558,27.020,154.736
C08042=1075.729,244.384,-83.283,174.560,27.024,154.736
C08043=1075.734,244.632,-83.310,174.562,27.028,154.737
C08044=1075.740,244.881,-83.337,174.566,27.032,154.737
C08045=1075.747,245.129,-83.364,174.568,27.036,154.738
C08046=1075.752,245.378,-83.391,174.570,27.039,154.738
C08047=1075.758,245.626,-83.418,174.572,27.043,154.739
C08048=1075.764,245.874,-83.446,174.575,27.047,154.740
C08049=1075.769,246.123,-83.473,174.577,27.050,154.740
C08050=1075.775,246.372,-83.500,174.580,27.054,154.741
C08051=1075.780,246.620,-83.528,174.582,27.058,154.741
C08052=1075.787,246.869,-83.555,174.585,27.062,154.742
C08053=1075.792,247.117,-83.583,174.587,27.065,154.742
C08054=1075.798,247.365,-83.609,174.589,27.069,154.743
C08055=1075.804,247.614,-83.637,174.591,27.073,154.743
C08056=1075.810,247.862,-83.664,174.595,27.077,154.744
C08057=1075.815,248.111,-83.692,174.597,27.081,154.745
C08058=1075.820,248.359,-83.720,174.599,27.085,154.745
C08059=1075.826,248.608,-83.747,174.601,27.089,154.746
C08060=1075.835,249.009,-83.791,174.605,27.095,154.747
C08061=1075.845,249.411,-83.836,174.610,27.101,154.748
C08062=1075.854,249.813,-83.880,174.614,27.107,154.749
C08063=1075.863,250.214,-83.925,174.617,27.113,154.749
C08064=1075.869,250.463,-83.953,174.620,27.117,154.750
C08065=1075.875,250.711,-83.980,174.622,27.121,154.751
C08066=1075.880,250.960,-84.008,174.624,27.124,154.751
C08067=1075.886,251.208,-84.036,174.627,27.129,154.752
C08068=1075.892,251.456,-84.062,174.630,27.132,154.752
C08069=1075.898,251.705,-84.091,174.632,27.136,154.753
C08070=1075.903,251.953,-84.119,174.634,27.140,154.753
C08071=1075.909,252.201,-84.145,174.637,27.143,154.754
C08072=1075.915,252.450,-84.174,174.640,27.148,154.755
C08073=1075.920,252.698,-84.202,174.642,27.151,154.755
C08074=1075.926,252.947,-84.229,174.644,27.155,154.756
C08075=1075.932,253.195,-84.257,174.647,27.159,154.756
C08076=1075.938,253.444,-84.285,174.650,27.163,154.757
C08077=1075.944,253.692,-84.312,174.652,27.167,154.757
C08078=1075.949,253.940,-84.340,174.654,27.170,154.758
C08079=1075.955,254.189,-84.368,174.657,27.174,154.759
C08080=1075.961,254.437,-84.395,174.659,27.178,154.759
C08081=1075.967,254.686,-84.424,174.662,27.182,154.760
C08082=1075.972,254.934,-84.452,174.664,27.185,154.760
C08083=1075.978,255.182,-84.480,174.667,27.189,154.761
C08084=1075.984,255.430,-84.507,174.669,27.193,154.761
C08085=1075.990,255.679,-84.535,174.672,27.197,154.762
C08086=1075.995,255.927,-84.563,174.674,27.201,154.763
C08087=1076.002,256.176,-84.591,174.677,27.204,154.763
C08088=1076.007,256.424,-84.619,174.679,27.208,154.764
C08089=1076.013,256.673,-84.647,174.682,27.212,154.764
C08090=1076.018,256.921,-84.675,174.685,27.216,154.765
C08091=1076.025,257.169,-84.703,174.687,27.220,154.765
C08092=1076.030,257.417,-84.731,174.689,27.223,154.766
C08093=1076.036,257.666,-84.759,174.692,27.227,154.766
C08094=1076.042,257.915,-84.787,174.695,27.231,154.767
C08095=1076.048,258.163,-84.815,174.697,27.234,154.768
C08096=1076.054,258.411,-84.843,174.699,27.238,154.768
C08097=1076.060,258.659,-84.871,174.702,27.242,154.769
C08098=1076.066,258.908,-84.899,174.705,27.246,154.769
C08099=1076.072,259.157,-84.927,174.707,27.249,154.770
C08100=1076.078,259.405,-84.955,174.709,27.253,154.770
C08101=1076.083,259.653,-84.983,174.712,27.257,154.771
C08102=1076.089,259.901,-85.011,174.715,27.261,154.771
C08103=1076.095,260.149,-85.040,174.717,27.264,154.772
C08104=1076.102,260.398,-85.068,174.720,27.269,154.773
C08105=1076.107,260.646,-85.096,174.723,27.272,154.773
C08106=1076.113,260.895,-85.124,174.725,27.276,154.774
C08107=1076.119,261.143,-85.152,174.727,27.280,154.774
C08108=1076.124,261.392,-85.180,174.730,27.283,154.775
C08109=1076.131,261.639,-85.209,174.733,27.287,154.775
C08110=1076.137,261.888,-85.237,174.735,27.291,154.776
C08111=1076.143,262.136,-85.265,174.738,27.295,154.776
C08112=1076.152,262.536,-85.311,174.742,27.300,154.777
C08113=1076.162,262.934,-85.356,174.746,27.307,154.778
C08114=1076.172,263.334,-85.402,174.750,27.312,154.779
C08115=1076.181,263.732,-85.448,174.755,27.319,154.780
C08116=1076.187,263.981,-85.476,174.757,27.322,154.781
C08117=1076.192,264.229,-85.504,174.759,27.326,154.781
C08118=1076.199,264.477,-85.533,174.763,27.330,154.782
C08119=1076.205,264.726,-85.561,174.765,27.334,154.782
C08120=1076.210,264.973,-85.590,174.767,27.338,154.783
C08121=1076.216,265.222,-85.619,174.770,27.342,154.783
C08122=1076.221,265.471,-85.647,174.773,27.346,154.784
C08123=1076.227,265.719,-85.676,174.775,27.349,154.785
C08124=1076.233,265.967,-85.704,174.777,27.353,154.785
C08125=1076.239,266.215,-85.733,174.780,27.357,154.786
C08126=1076.245,266.464,-85.762,174.783,27.361,154.786
C08127=1076.251,266.712,-85.790,174.785,27.364,154.787
C08128=1076.257,266.960,-85.819,174.788,27.369,154.788
C08129=1076.262,267.209,-85.848,174.791,27.372,154.788
C08130=1076.268,267.457,-85.876,174.793,27.376,154.789
C08131=1076.274,267.705,-85.905,174.796,27.380,154.789
C08132=1076.280,267.954,-85.934,174.798,27.384,154.790
C08133=1076.286,268.202,-85.963,174.801,27.388,154.790
C08134=1076.292,268.449,-85.991,174.804,27.391,154.791
C08135=1076.297,268.698,-86.020,174.806,27.395,154.792
C08136=1076.303,268.946,-86.049,174.808,27.399,154.792
C08137=1076.309,269.195,-86.078,174.812,27.403,154.793
C08138=1076.315,269.443,-86.107,174.814,27.407,154.793
C08139=1076.320,269.691,-86.136,174.816,27.411,154.794
C08140=1076.327,269.939,-86.165,174.820,27.414,154.794
C08141=1076.333,270.188,-86.193,174.822,27.419,154.795
C08142=1076.339,270.436,-86.222,174.824,27.422,154.796
C08143=1076.344,270.685,-86.252,174.827,27.426,154.796
C08144=1076.350,270.933,-86.280,174.830,27.430,154.797
C08145=1076.356,271.181,-86.309,174.832,27.434,154.797
C08146=1076.361,271.429,-86.339,174.835,27.438,154.798
C08147=1076.368,271.677,-86.368,174.837,27.442,154.799
C08148=1076.374,271.925,-86.397,174.841,27.445,154.799
C08149=1076.378,272.174,-86.425,174.843,27.449,154.800
C08150=1076.385,272.422,-86.454,174.845,27.453,154.800
C08151=1076.391,272.670,-86.483,174.849,27.457,154.801
C08152=1076.396,272.919,-86.513,174.851,27.461,154.801
C08153=1076.403,273.167,-86.542,174.853,27.465,154.802
C08154=1076.409,273.415,-86.571,174.856,27.469,154.803
C08155=1076.415,273.663,-86.601,174.859,27.473,154.803
C08156=1076.420,273.911,-86.629,174.861,27.476,154.804
C08157=1076.425,274.160,-86.658,174.864,27.480,154.804
C08158=1076.432,274.408,-86.687,174.867,27.484,154.805
C08159=1076.437,274.656,-86.717,174.870,27.488,154.806
C08160=1076.443,274.904,-86.746,174.872,27.492,154.806
C08161=1076.449,275.153,-86.776,174.874,27.496,154.807
C08162=1076.455,275.401,-86.805,174.878,27.499,154.807
C08163=1076.461,275.649,-86.834,174.880,27.503,154.808
C08164=1076.470,276.051,-86.882,174.885,27.510,154.809
C08165=1076.479,276.453,-86.929,174.889,27.516,154.810
C08166=1076.489,276.856,-86.977,174.893,27.522,154.811
C08167=1076.499,277.257,-87.025,174.897,27.529,154.812
C08168=1076.504,277.506,-87.054,174.900,27.533,154.812
C08169=1076.510,277.754,-87.083,174.903,27.536,154.813
C08170=1076.516,278.002,-87.113,174.905,27.540,154.814
C08171=1076.522,278.251,-87.142,174.908,27.545,154.814
C08172=1076.528,278.498,-87.172,174.911,27.548,154.815
C08173=1076.534,278.746,-87.202,174.913,27.552,154.815
C08174=1076.540,278.995,-87.231,174.916,27.556,154.816
C08175=1076.545,279.243,-87.261,174.918,27.560,154.817
C08176=1076.551,279.491,-87.290,174.922,27.564,154.817
C08177=1076.557,279.739,-87.320,174.924,27.568,154.818
C08178=1076.563,279.988,-87.350,174.927,27.572,154.818
C08179=1076.569,280.236,-87.379,174.930,27.575,154.819
C08180=1076.575,280.484,-87.409,174.932,27.579,154.819
C08181=1076.581,280.732,-87.438,174.935,27.583,154.820
C08182=1076.587,280.980,-87.468,174.937,27.587,154.821
C08183=1076.592,281.228,-87.498,174.941,27.591,154.821
C08184=1076.598,281.477,-87.528,174.943,27.595,154.822
C08185=1076.603,281.725,-87.558,174.946,27.599,154.822
C08186=1076.610,281.972,-87.587,174.949,27.603,154.823
C08187=1076.615,282.221,-87.617,174.951,27.607,154.824
C08188=1076.621,282.469,-87.647,174.954,27.611,154.824
C08189=1076.627,282.717,-87.677,174.956,27.615,154.825
C08190=1076.632,282.966,-87.707,174.960,27.619,154.826
C08191=1076.639,283.213,-87.736,174.962,27.623,154.826
C08192=1076.644,283.462,-87.766,174.965,27.627,154.827
C08193=1076.650,283.709,-87.796,174.967,27.631,154.827
C08194=1076.656,283.958,-87.826,174.971,27.635,154.828
C08195=1076.662,284.206,-87.856,174.973,27.639,154.829
C08196=1076.667,284.453,-87.887,174.975,27.643,154.829
C08197=1076.674,284.702,-87.916,174.979,27.647,154.830
C08198=1076.679,284.949,-87.946,174.981,27.650,154.830
C08199=1076.685,285.198,-87.976,174.984,27.655,154.831
C08200=1076.691,285.446,-88.006,174.986,27.659,154.832
C08201=1076.697,285.695,-88.036,174.990,27.663,154.832
C08202=1076.703,285.943,-88.066,174.992,27.666,154.833
C08203=1076.708,286.190,-88.097,174.995,27.671,154.833
C08204=1076.715,286.439,-88.126,174.998,27.675,154.834
C08205=1076.721,286.686,-88.156,175.001,27.678,154.835
C08206=1076.726,286.934,-88.186,175.003,27.682,154.835
C08207=1076.732,287.183,-88.216,175.006,27.687,154.836
C08208=1076.738,287.431,-88.247,175.009,27.691,154.837
C08209=1076.744,287.679,-88.277,175.012,27.694,154.837
C08210=1076.750,287.927,-88.307,175.014,27.698,154.838
C08211=1076.755,288.175,-88.337,175.017,27.703,154.838
C08212=1076.761,288.423,-88.367,175.020,27.706,154.839
C08213=1076.768,288.672,-88.398,175.022,27.710,154.840
C08214=1076.774,288.919,-88.428,175.025,27.714,154.840
C08215=1076.780,289.167,-88.458,175.028,27.718,154.841
C08216=1076.790,289.580,-88.509,175.032,27.725,154.842
C08217=1076.799,289.991,-88.559,175.037,27.732,154.843
C08218=1076.809,290.404,-88.609,175.042,27.739,154.844
C08219=1076.819,290.816,-88.660,175.047,27.745,154.845
C08220=1076.825,291.064,-88.691,175.049,27.749,154.846
C08221=1076.831,291.311,-88.721,175.052,27.753,154.846
C08222=1076.835,291.560,-88.751,175.055,27.757,154.847
C08223=1076.842,291.809,-88.782,175.058,27.761,154.847
C08224=1076.848,292.057,-88.812,175.060,27.765,154.848
C08225=1076.854,292.304,-88.843,175.064,27.769,154.849
C08226=1076.860,292.552,-88.874,175.066,27.773,154.849
C08227=1076.866,292.800,-88.905,175.069,27.777,154.850
C08228=1076.872,293.048,-88.935,175.071,27.781,154.851
C08229=1076.877,293.296,-88.966,175.075,27.786,154.851
C08230=1076.883,293.544,-88.996,175.077,27.790,154.852
C08231=1076.889,293.792,-89.027,175.080,27.794,154.853
C08232=1076.895,294.040,-89.057,175.083,27.798,154.853
C08233=1076.901,294.288,-89.088,175.086,27.802,154.854
C08234=1076.906,294.537,-89.119,175.089,27.806,154.854
C08235=1076.913,294.784,-89.150,175.091,27.810,154.855
C08236=1076.918,295.032,-89.180,175.095,27.814,154.856
C08237=1076.925,295.280,-89.211,175.097,27.818,154.856
C08238=1076.931,295.528,-89.241,175.100,27.822,154.857
C08239=1076.936,295.776,-89.272,175.102,27.826,154.858
C08240=1076.942,296.024,-89.304,175.106,27.830,154.858
C08241=1076.948,296.272,-89.334,175.108,27.834,154.859
C08242=1076.953,296.520,-89.365,175.111,27.839,154.859
C08243=1076.960,296.769,-89.396,175.114,27.843,154.860
C08244=1076.966,297.016,-89.427,175.117,27.847,154.861
C08245=1076.971,297.264,-89.458,175.120,27.851,154.861
C08246=1076.977,297.513,-89.489,175.122,27.855,154.862
C08247=1076.984,297.760,-89.520,175.126,27.859,154.863
C08248=1076.989,298.008,-89.551,175.128,27.863,154.863
C08249=1076.995,298.256,-89.582,175.131,27.868,154.864
C08250=1077.000,298.504,-89.613,175.134,27.872,154.865
C08251=1077.006,298.752,-89.643,175.137,27.876,154.865
C08252=1077.012,299.000,-89.675,175.140,27.880,154.866
C08253=1077.017,299.248,-89.706,175.142,27.884,154.867
C08254=1077.023,299.495,-89.737,175.145,27.889,154.867
C08255=1077.029,299.744,-89.769,175.148,27.893,154.868
C08256=1077.035,299.991,-89.800,175.151,27.897,154.869
C08257=1077.041,300.240,-89.831,175.154,27.901,154.869
C08258=1077.047,300.487,-89.862,175.157,27.905,154.870
C08259=1077.052,300.736,-89.893,175.160,27.909,154.871
C08260=1077.058,300.984,-89.925,175.162,27.913,154.871
C08261=1077.064,301.231,-89.956,175.165,27.918,154.872
C08262=1077.069,301.479,-89.987,175.169,27.922,154.873
C08263=1077.076,301.727,-90.018,175.171,27.926,154.873
C08264=1077.081,301.975,-90.049,175.174,27.930,154.874
C08265=1077.087,302.223,-90.081,175.177,27.934,154.875
C08266=1077.093,302.471,-90.112,175.180,27.939,154.875
C08267=1077.099,302.719,-90.144,175.183,27.943,154.876
C08268=1077.103,302.932,-90.171,175.185,27.947,154.877
C08269=1077.109,303.146,-90.197,175.188,27.950,154.877
C08270=1077.114,303.359,-90.225,175.190,27.954,154.878
C08271=1077.119,303.572,-90.253,175.192,27.958,154.878
C08272=1077.124,303.785,-90.279,175.195,27.961,154.879
C08273=1077.129,303.998,-90.306,175.197,27.965,154.880
C08274=1077.134,304.212,-90.333,175.200,27.968,154.880
C08275=1077.139,304.425,-90.361,175.203,27.972,154.881
C08276=1077.145,304.673,-90.392,175.205,27.977,154.881
C08277=1077.151,304.922,-90.423,175.208,27.981,154.882
C08278=1077.156,305.169,-90.455,175.212,27.985,154.883
C08279=1077.163,305.417,-90.486,175.214,27.989,154.883
C08280=1077.168,305.664,-90.518,175.217,27.994,154.884
C08281=1077.174,305.913,-90.550,175.220,27.998,154.885
C08282=1077.181,306.160,-90.581,175.223,28.002,154.885
C08283=1077.187,306.408,-90.613,175.226,28.006,154.886
C08284=1077.193,306.656,-90.645,175.228,28.010,154.887
C08285=1077.198,306.904,-90.677,175.232,28.015,154.887
C08286=1077.204,307.152,-90.707,175.235,28.019,154.888
C08287=1077.210,307.400,-90.739,175.237,28.023,154.889
C08288=1077.216,307.648,-90.771,175.241,28.027,154.889
C08289=1077.222,307.896,-90.803,175.244,28.032,154.890
C08290=1077.228,308.143,-90.834,175.246,28.036,154.891
C08291=1077.234,308.392,-90.866,175.249,28.040,154.891
C08292=1077.240,308.639,-90.899,175.253,28.045,154.892
C08293=1077.246,308.886,-90.930,175.255,28.049,154.893
C08294=1077.252,309.135,-90.962,175.258,28.053,154.893
C08295=1077.258,309.383,-90.994,175.261,28.057,154.894
C08296=1077.264,309.630,-91.026,175.264,28.062,154.895
C08297=1077.270,309.878,-91.057,175.267,28.066,154.896
C08298=1077.276,310.127,-91.089,175.270,28.070,154.896
C08299=1077.282,310.374,-91.121,175.274,28.074,154.897
C08300=1077.288,310.622,-91.153,175.276,28.079,154.898
C08301=1077.294,310.870,-91.186,175.279,28.083,154.898
C08302=1077.300,311.117,-91.217,175.282,28.087,154.899
C08303=1077.306,311.365,-91.249,175.285,28.091,154.900
C08304=1077.312,311.613,-91.281,175.288,28.096,154.900
C08305=1077.318,311.862,-91.313,175.291,28.100,154.901
C08306=1077.324,312.109,-91.346,175.293,28.104,154.902
C08307=1077.330,312.356,-91.377,175.297,28.109,154.902
C08308=1077.336,312.605,-91.409,175.300,28.113,154.903
C08309=1077.342,312.853,-91.441,175.303,28.117,154.904
C08310=1077.349,313.100,-91.473,175.306,28.121,154.904
C08311=1077.355,313.349,-91.505,175.309,28.126,154.905
C08312=1077.360,313.596,-91.537,175.312,28.130,154.906
C08313=1077.367,313.843,-91.569,175.314,28.134,154.907
C08314=1077.373,314.092,-91.601,175.318,28.138,154.907
C08315=1077.379,314.339,-91.634,175.321,28.143,154.908
C08316=1077.385,314.588,-91.666,175.324,28.147,154.909
C08317=1077.391,314.836,-91.698,175.326,28.152,154.909
C08318=1077.397,315.083,-91.730,175.330,28.156,154.910
C08319=1077.402,315.331,-91.763,175.333,28.161,154.911
C08320=1077.409,315.579,-91.796,175.335,28.165,154.912
C08321=1077.415,315.827,-91.828,175.338,28.170,154.912
C08322=1077.420,316.074,-91.861,175.342,28.174,154.913
C08323=1077.426,316.322,-91.893,175.345,28.179,154.914
C08324=1077.430,316.537,-91.921,175.347,28.183,154.914
C08325=1077.436,316.752,-91.950,175.350,28.187,154.915
C08326=1077.441,316.967,-91.978,175.352,28.190,154.916
C08327=1077.446,317.181,-92.006,175.355,28.194,154.916
C08328=1077.452,317.397,-92.034,175.358,28.198,154.917
C08329=1077.456,317.611,-92.062,175.360,28.202,154.918
C08330=1077.461,317.826,-92.091,175.362,28.206,154.918
C08331=1077.467,318.041,-92.119,175.365,28.210,154.919
C08332=1077.473,318.289,-92.151,175.368,28.215,154.920
C08333=1077.478,318.537,-92.184,175.371,28.219,154.920
C08334=1077.484,318.784,-92.217,175.375,28.223,154.921
C08335=1077.490,319.032,-92.249,175.377,28.228,154.922
C08336=1077.495,319.280,-92.282,175.380,28.233,154.923
C08337=1077.502,319.528,-92.315,175.383,28.237,154.923
C08338=1077.508,319.776,-92.348,175.387,28.241,154.924
C08339=1077.513,320.024,-92.380,175.390,28.246,154.925
C08340=1077.519,320.272,-92.413,175.392,28.251,154.926
C08341=1077.525,320.520,-92.446,175.395,28.255,154.926
C08342=1077.531,320.767,-92.479,175.399,28.259,154.927
C08343=1077.537,321.014,-92.512,175.402,28.264,154.928
C08344=1077.543,321.262,-92.545,175.404,28.269,154.929
C08345=1077.549,321.510,-92.577,175.407,28.273,154.929
C08346=1077.555,321.758,-92.610,175.411,28.278,154.930
C08347=1077.560,322.006,-92.643,175.414,28.283,154.931
C08348=1077.567,322.253,-92.676,175.417,28.287,154.932
C08349=1077.572,322.501,-92.709,175.420,28.291,154.932
C08350=1077.579,322.749,-92.742,175.423,28.296,154.933
C08351=1077.585,322.996,-92.775,175.426,28.301,154.934
C08352=1077.590,323.244,-92.808,175.429,28.305,154.935
C08353=1077.597,323.492,-92.841,175.432,28.310,154.935
C08354=1077.602,323.740,-92.874,175.435,28.314,154.936
C08355=1077.609,323.987,-92.907,175.438,28.319,154.937
C08356=1077.615,324.236,-92.940,175.441,28.324,154.938
C08357=1077.621,324.484,-92.973,175.444,28.328,154.939
C08358=1077.627,324.731,-93.007,175.448,28.333,154.939
C08359=1077.633,324.979,-93.039,175.450,28.337,154.940
C08360=1077.639,325.227,-93.072,175.453,28.342,154.941
C08361=1077.645,325.475,-93.105,175.457,28.346,154.942
C08362=1077.651,325.722,-93.139,175.460,28.351,154.942
C08363=1077.657,325.969,-93.172,175.463,28.356,154.943
C08364=1077.663,326.217,-93.205,175.466,28.360,154.944
C08365=1077.669,326.465,-93.238,175.469,28.365,154.945
C08366=1077.676,326.713,-93.271,175.472,28.369,154.945
C08367=1077.681,326.961,-93.305,175.475,28.374,154.946
C08368=1077.688,327.208,-93.338,175.478,28.379,154.947
C08369=1077.693,327.456,-93.371,175.482,28.383,154.948
C08370=1077.700,327.704,-93.404,175.485,28.388,154.949
C08371=1077.705,327.951,-93.438,175.488,28.393,154.949
C08372=1077.712,328.199,-93.471,175.490,28.397,154.950
C08373=1077.718,328.447,-93.505,175.494,28.402,154.951
C08374=1077.724,328.694,-93.538,175.497,28.407,154.952
C08375=1077.730,328.942,-93.572,175.500,28.411,154.952
C08376=1077.736,329.191,-93.605,175.503,28.416,154.953
C08377=1077.743,329.438,-93.639,175.507,28.421,154.954
C08378=1077.748,329.685,-93.672,175.510,28.426,154.955
C08379=1077.755,329.933,-93.705,175.513,28.430,154.956
C08380=1077.761,330.145,-93.734,175.516,28.434,154.956
C08381=1077.765,330.356,-93.762,175.518,28.438,154.957
C08382=1077.770,330.568,-93.791,175.520,28.442,154.958
C08383=1077.776,330.780,-93.820,175.524,28.446,154.958
C08384=1077.781,330.991,-93.849,175.526,28.450,154.959
C08385=1077.786,331.203,-93.877,175.528,28.454,154.960
C08386=1077.792,331.415,-93.906,175.532,28.458,154.960
C08387=1077.797,331.626,-93.935,175.534,28.462,154.961
C08388=1077.803,331.874,-93.969,175.537,28.467,154.962
C08389=1077.809,332.122,-94.002,175.541,28.472,154.963
C08390=1077.815,332.370,-94.036,175.544,28.477,154.963
C08391=1077.821,332.617,-94.070,175.547,28.482,154.964
C08392=1077.827,332.864,-94.103,175.550,28.486,154.965
C08393=1077.833,333.112,-94.137,175.554,28.492,154.966
C08394=1077.839,333.360,-94.171,175.556,28.496,154.967
C08395=1077.845,333.608,-94.205,175.559,28.501,154.968
C08396=1077.851,333.855,-94.239,175.562,28.506,154.968
C08397=1077.857,334.103,-94.274,175.566,28.510,154.969
C08398=1077.863,334.351,-94.307,175.569,28.516,154.970
C08399=1077.869,334.598,-94.341,175.572,28.520,154.971
C08400=1077.875,334.845,-94.375,175.575,28.525,154.972
C08401=1077.881,335.093,-94.409,175.579,28.530,154.973
C08402=1077.887,335.341,-94.442,175.582,28.535,154.973
C08403=1077.894,335.589,-94.477,175.585,28.540,154.974
C08404=1077.900,335.836,-94.511,175.588,28.545,154.975
C08405=1077.906,336.083,-94.545,175.591,28.550,154.976
C08406=1077.912,336.331,-94.579,175.595,28.555,154.977
C08407=1077.918,336.579,-94.613,175.598,28.559,154.978
C08408=1077.924,336.826,-94.647,175.601,28.565,154.978
C08409=1077.930,337.074,-94.682,175.604,28.570,154.979
C08410=1077.936,337.321,-94.716,175.608,28.574,154.980
C08411=1077.942,337.570,-94.749,175.611,28.580,154.981
C08412=1077.948,337.817,-94.783,175.614,28.584,154.982
C08413=1077.955,338.065,-94.818,175.617,28.589,154.983
C08414=1077.960,338.312,-94.852,175.620,28.594,154.984
C08415=1077.967,338.559,-94.887,175.623,28.599,154.985
C08416=1077.972,338.807,-94.922,175.626,28.604,154.985
C08417=1077.978,339.055,-94.956,175.629,28.609,154.986
C08418=1077.985,339.303,-94.990,175.633,28.614,154.987
C08419=1077.990,339.550,-95.024,175.636,28.619,154.988
C08420=1077.996,339.797,-95.058,175.639,28.624,154.989
C08421=1078.003,340.045,-95.093,175.642,28.629,154.990
C08422=1078.008,340.293,-95.127,175.645,28.634,154.991
C08423=1078.015,340.540,-95.162,175.649,28.640,154.991
C08424=1078.021,340.787,-95.197,175.652,28.645,154.992
C08425=1078.027,341.035,-95.231,175.655,28.650,154.993
C08426=1078.033,341.283,-95.265,175.658,28.655,154.994
C08427=1078.039,341.531,-95.300,175.662,28.660,154.995
C08428=1078.045,341.778,-95.335,175.665,28.665,154.996
C08429=1078.051,342.026,-95.369,175.668,28.670,154.997
C08430=1078.057,342.273,-95.403,175.671,28.675,154.998
C08431=1078.064,342.520,-95.438,175.675,28.680,154.999
C08432=1078.070,342.769,-95.473,175.679,28.686,154.999
C08433=1078.075,343.016,-95.507,175.682,28.691,155.000
C08434=1078.082,343.263,-95.543,175.685,28.696,155.001
C08435=1078.088,343.511,-95.577,175.688,28.701,155.002
C08436=1078.098,343.929,-95.636,175.694,28.709,155.004
C08437=1078.109,344.347,-95.695,175.699,28.718,155.005
C08438=1078.119,344.765,-95.753,175.705,28.727,155.007
C08439=1078.129,345.183,-95.812,175.710,28.736,155.008
C08440=1078.136,345.430,-95.847,175.713,28.741,155.009
C08441=1078.142,345.677,-95.882,175.717,28.746,155.010
C08442=1078.148,345.925,-95.917,175.720,28.751,155.011
C08443=1078.153,346.172,-95.951,175.723,28.757,155.012
C08444=1078.159,346.420,-95.987,175.726,28.762,155.013
C08445=1078.166,346.667,-96.022,175.730,28.767,155.014
C08446=1078.171,346.915,-96.057,175.734,28.773,155.015
C08447=1078.178,347.162,-96.092,175.737,28.778,155.016
C08448=1078.184,347.410,-96.128,175.740,28.783,155.017
C08449=1078.190,347.657,-96.162,175.743,28.789,155.018
C08450=1078.196,347.905,-96.197,175.747,28.794,155.019
C08451=1078.203,348.152,-96.233,175.750,28.799,155.020
C08452=1078.208,348.399,-96.268,175.753,28.804,155.020
C08453=1078.215,348.647,-96.302,175.756,28.810,155.021
C08454=1078.221,348.895,-96.338,175.760,28.815,155.022
C08455=1078.227,349.142,-96.373,175.763,28.820,155.023
C08456=1078.233,349.389,-96.409,175.767,28.826,155.024
C08457=1078.239,349.637,-96.444,175.770,28.831,155.025
C08458=1078.246,349.884,-96.480,175.773,28.837,155.026
C08459=1078.251,350.131,-96.515,175.777,28.842,155.027
C08460=1078.258,350.379,-96.549,175.780,28.848,155.028
C08461=1078.264,350.627,-96.585,175.783,28.853,155.029
C08462=1078.270,350.874,-96.620,175.786,28.858,155.030
C08463=1078.276,351.121,-96.656,175.789,28.863,155.031
C08464=1078.282,351.369,-96.691,175.794,28.869,155.032
C08465=1078.289,351.616,-96.726,175.797,28.874,155.033
C08466=1078.295,351.864,-96.762,175.800,28.880,155.034
C08467=1078.301,352.112,-96.798,175.803,28.885,155.035
C08468=1078.307,352.358,-96.833,175.807,28.891,155.036
C08469=1078.313,352.605,-96.869,175.810,28.896,155.037
C08470=1078.319,352.853,-96.905,175.814,28.902,155.038
C08471=1078.326,353.100,-96.940,175.817,28.907,155.039
C08472=1078.332,353.348,-96.976,175.820,28.913,155.040
C08473=1078.337,353.595,-97.011,175.824,28.919,155.041
C08474=1078.343,353.843,-97.047,175.827,28.924,155.042
C08475=1078.350,354.090,-97.083,175.830,28.929,155.043
C08476=1078.357,354.337,-97.118,175.834,28.935,155.044
C08477=1078.363,354.585,-97.154,175.837,28.941,155.045
C08478=1078.369,354.832,-97.190,175.841,28.946,155.046
C08479=1078.375,355.080,-97.226,175.844,28.952,155.047
C08480=1078.380,355.326,-97.262,175.847,28.957,155.048
C08481=1078.386,355.574,-97.297,175.850,28.963,155.049
C08482=1078.394,355.821,-97.333,175.854,28.969,155.050
C08483=1078.400,356.069,-97.369,175.858,28.975,155.051
C08484=1078.406,356.316,-97.405,175.861,28.980,155.052
C08485=1078.412,356.563,-97.441,175.864,28.986,155.053
C08486=1078.418,356.811,-97.477,175.868,28.992,155.054
C08487=1078.424,357.058,-97.513,175.871,28.997,155.055
C08488=1078.429,357.269,-97.544,175.874,29.002,155.056
C08489=1078.435,357.479,-97.573,175.877,29.007,155.057
C08490=1078.440,357.690,-97.605,175.880,29.012,155.058
C08491=1078.445,357.901,-97.635,175.883,29.016,155.059
C08492=1078.450,358.111,-97.666,175.886,29.021,155.059
C08493=1078.456,358.322,-97.697,175.888,29.026,155.060
C08494=1078.462,358.532,-97.727,175.892,29.031,155.061
C08495=1078.467,358.743,-97.758,175.895,29.036,155.062
C08496=1078.473,358.990,-97.794,175.898,29.042,155.063
C08497=1078.479,359.237,-97.830,175.901,29.047,155.064
C08498=1078.485,359.484,-97.866,175.905,29.053,155.065
C08499=1078.492,359.731,-97.903,175.909,29.059,155.066
C08500=1078.498,359.979,-97.939,175.912,29.065,155.068
C08501=1078.504,360.226,-97.975,175.915,29.070,155.069
C08502=1078.510,360.473,-98.011,175.918,29.076,155.070
C08503=1078.517,360.720,-98.048,175.923,29.082,155.071
C08504=1078.522,360.968,-98.084,175.926,29.088,155.072
C08505=1078.528,361.215,-98.121,175.929,29.094,155.073
C08506=1078.535,361.462,-98.157,175.932,29.099,155.074
C08507=1078.541,361.709,-98.194,175.936,29.106,155.075
C08508=1078.548,361.957,-98.230,175.940,29.111,155.076
C08509=1078.554,362.205,-98.266,175.943,29.117,155.077
C08510=1078.560,362.452,-98.303,175.946,29.123,155.078
C08511=1078.567,362.699,-98.339,175.950,29.129,155.079
C08512=1078.573,362.946,-98.375,175.953,29.135,155.080
C08513=1078.579,363.193,-98.413,175.957,29.141,155.082
C08514=1078.585,363.440,-98.449,175.961,29.147,155.083
C08515=1078.591,363.687,-98.485,175.964,29.153,155.084
C08516=1078.598,363.934,-98.522,175.967,29.159,155.085
C08517=1078.605,364.182,-98.559,175.971,29.165,155.086
C08518=1078.611,364.429,-98.595,175.975,29.171,155.087
C08519=1078.617,364.677,-98.632,175.978,29.177,155.088
C08520=1078.623,364.924,-98.669,175.982,29.183,155.089
C08521=1078.629,365.171,-98.705,175.985,29.189,155.091
C08522=1078.636,365.418,-98.741,175.988,29.195,155.092
C08523=1078.641,365.665,-98.779,175.993,29.201,155.093
C08524=1078.648,365.912,-98.816,175.996,29.207,155.094
C08525=1078.654,366.160,-98.853,175.999,29.213,155.095
C08526=1078.660,366.407,-98.890,176.003,29.219,155.096
C08527=1078.667,366.654,-98.926,176.006,29.225,155.097
C08528=1078.673,366.901,-98.964,176.009,29.232,155.099
C08529=1078.679,367.148,-99.000,176.014,29.238,155.100
C08530=1078.685,367.396,-99.038,176.017,29.244,155.101
C08531=1078.691,367.643,-99.074,176.020,29.250,155.102
C08532=1078.697,367.889,-99.112,176.024,29.257,155.103
C08533=1078.704,368.136,-99.148,176.027,29.263,155.104
C08534=1078.711,368.384,-99.186,176.031,29.269,155.106
C08535=1078.716,368.631,-99.223,176.035,29.275,155.107
C08536=1078.723,368.878,-99.259,176.038,29.281,155.108
C08537=1078.729,369.125,-99.297,176.042,29.288,155.109
C08538=1078.736,369.373,-99.334,176.045,29.294,155.110
C08539=1078.742,369.619,-99.372,176.048,29.300,155.112
C08540=1078.748,369.866,-99.408,176.053,29.306,155.113
C08541=1078.754,370.113,-99.446,176.056,29.313,155.114
C08542=1078.761,370.361,-99.483,176.059,29.319,155.115
C08543=1078.767,370.608,-99.520,176.063,29.325,155.116
C08544=1078.773,370.826,-99.553,176.066,29.331,155.117
C08545=1078.778,371.045,-99.586,176.070,29.337,155.118
C08546=1078.784,371.263,-99.619,176.073,29.342,155.120
C08547=1078.789,371.483,-99.652,176.076,29.348,155.121
C08548=1078.795,371.701,-99.685,176.079,29.353,155.122
C08549=1078.801,371.920,-99.719,176.082,29.359,155.123
C08550=1078.807,372.138,-99.751,176.085,29.365,155.124
C08551=1078.812,372.357,-99.784,176.088,29.370,155.125
C08552=1078.818,372.604,-99.822,176.093,29.377,155.126
C08553=1078.825,372.851,-99.859,176.096,29.383,155.127
C08554=1078.831,373.099,-99.897,176.100,29.390,155.129
C08555=1078.838,373.345,-99.934,176.103,29.396,155.130
C08556=1078.844,373.593,-99.972,176.106,29.402,155.131
C08557=1078.851,373.839,-100.009,176.111,29.409,155.132
C08558=1078.857,374.086,-100.047,176.114,29.416,155.134
C08559=1078.863,374.334,-100.085,176.118,29.422,155.135
C08560=1078.869,374.581,-100.122,176.121,29.429,155.136
C08561=1078.875,374.828,-100.160,176.125,29.436,155.137
C08562=1078.882,375.075,-100.198,176.128,29.442,155.139
C08563=1078.888,375.321,-100.235,176.133,29.448,155.140
C08564=1078.895,375.569,-100.273,176.136,29.455,155.141
C08565=1078.900,375.816,-100.311,176.140,29.462,155.142
C08566=1078.907,376.063,-100.349,176.143,29.469,155.144
C08567=1078.914,376.309,-100.387,176.147,29.476,155.145
C08568=1078.920,376.557,-100.425,176.150,29.482,155.146
C08569=1078.926,376.803,-100.463,176.155,29.489,155.148
C08570=1078.933,377.051,-100.501,176.158,29.495,155.149
C08571=1078.939,377.297,-100.539,176.162,29.502,155.150
C08572=1078.945,377.545,-100.577,176.165,29.509,155.152
C08573=1078.951,377.791,-100.615,176.169,29.516,155.153
C08574=1078.958,378.039,-100.652,176.172,29.522,155.154
C08575=1078.965,378.285,-100.691,176.177,29.529,155.155
C08576=1078.971,378.532,-100.729,176.180,29.536,155.157
C08577=1078.977,378.779,-100.767,176.184,29.543,155.158
C08578=1078.983,379.026,-100.805,176.187,29.549,155.159
C08579=1078.990,379.273,-100.844,176.191,29.556,155.161
C08580=1078.996,379.520,-100.881,176.194,29.563,155.162
C08581=1079.003,379.767,-100.920,176.199,29.570,155.163
C08582=1079.010,380.013,-100.957,176.202,29.577,155.165
C08583=1079.016,380.261,-100.996,176.206,29.584,155.166
C08584=1079.023,380.507,-101.034,176.210,29.591,155.168
C08585=1079.029,380.754,-101.072,176.213,29.597,155.169
C08586=1079.036,381.001,-101.111,176.218,29.605,155.170
C08587=1079.042,381.248,-101.149,176.221,29.611,155.172
C08588=1079.048,381.495,-101.188,176.225,29.618,155.173
C08589=1079.055,381.742,-101.226,176.228,29.625,155.174
C08590=1079.062,381.989,-101.265,176.232,29.632,155.176
C08591=1079.068,382.236,-101.303,176.236,29.639,155.177
C08592=1079.074,382.482,-101.341,176.240,29.646,155.178
C08593=1079.081,382.729,-101.380,176.244,29.653,155.180
C08594=1079.086,382.976,-101.418,176.247,29.660,155.181
C08595=1079.093,383.223,-101.457,176.251,29.668,155.183
C08596=1079.100,383.470,-101.496,176.255,29.675,155.184
C08597=1079.106,383.717,-101.534,176.258,29.682,155.185
C08598=1079.113,383.963,-101.573,176.263,29.689,155.187
C08599=1079.119,384.211,-101.612,176.267,29.696,155.188
C08600=1079.125,384.444,-101.649,176.270,29.703,155.190
C08601=1079.132,384.676,-101.685,176.273,29.710,155.191
C08602=1079.137,384.910,-101.721,176.277,29.717,155.192
C08603=1079.144,385.143,-101.758,176.281,29.723,155.194
C08604=1079.150,385.376,-101.795,176.284,29.730,155.195
C08605=1079.156,385.609,-101.832,176.288,29.738,155.197
C08606=1079.162,385.842,-101.869,176.291,29.744,155.198
C08607=1079.168,386.075,-101.905,176.295,29.751,155.199
C08608=1079.174,386.321,-101.944,176.299,29.758,155.201
C08609=1079.181,386.568,-101.983,176.303,29.766,155.202
C08610=1079.187,386.815,-102.022,176.307,29.773,155.204
C08611=1079.194,387.062,-102.061,176.310,29.781,155.205
C08612=1079.201,387.309,-102.100,176.314,29.788,155.207
C08613=1079.207,387.556,-102.139,176.318,29.795,155.208
C08614=1079.213,387.803,-102.178,176.322,29.802,155.209
C08615=1079.220,388.049,-102.217,176.326,29.810,155.211
C08616=1079.226,388.296,-102.255,176.330,29.817,155.212
C08617=1079.233,388.543,-102.295,176.334,29.825,155.214
C08618=1079.240,388.789,-102.334,176.337,29.832,155.215
C08619=1079.246,389.036,-102.373,176.341,29.840,155.217
C08620=1079.253,389.283,-102.413,176.346,29.847,155.218
C08621=1079.259,389.530,-102.452,176.349,29.855,155.220
C08622=1079.266,389.776,-102.491,176.353,29.862,155.222
C08623=1079.273,390.023,-102.530,176.357,29.870,155.223
C08624=1079.279,390.270,-102.569,176.361,29.878,155.225
C08625=1079.286,390.516,-102.609,176.364,29.885,155.226
C08626=1079.293,390.763,-102.648,176.369,29.893,155.228
C08627=1079.299,391.010,-102.687,176.373,29.900,155.229
C08628=1079.306,391.257,-102.727,176.377,29.908,155.231
C08629=1079.313,391.504,-102.766,176.381,29.916,155.232
C08630=1079.319,391.750,-102.806,176.384,29.923,155.234
C08631=1079.326,391.997,-102.845,176.388,29.931,155.235
C08632=1079.332,392.243,-102.885,176.393,29.939,155.237
C08633=1079.339,392.490,-102.924,176.397,29.947,155.239
C08634=1079.345,392.737,-102.964,176.400,29.954,155.240
C08635=1079.352,392.984,-103.003,176.404,29.962,155.242
C08636=1079.359,393.230,-103.043,176.408,29.970,155.243
C08637=1079.365,393.477,-103.083,176.412,29.978,155.245
C08638=1079.372,393.723,-103.122,176.417,29.986,155.246
C08639=1079.379,393.971,-103.163,176.420,29.994,155.248
C08640=1079.385,394.217,-103.203,176.424,30.001,155.250
C08641=1079.392,394.463,-103.242,176.428,30.009,155.251
C08642=1079.398,394.710,-103.282,176.432,30.018,155.253
C08643=1079.405,394.957,-103.322,176.436,30.025,155.255
C08644=1079.412,395.203,-103.362,176.440,30.033,155.256
C08645=1079.418,395.450,-103.402,176.444,30.041,155.258
C08646=1079.425,395.697,-103.442,176.448,30.049,155.260
C08647=1079.431,395.944,-103.482,176.452,30.058,155.261
C08648=1079.438,396.191,-103.522,176.456,30.066,155.263
C08649=1079.445,396.437,-103.561,176.460,30.074,155.265
C08650=1079.451,396.683,-103.602,176.465,30.082,155.266
C08651=1079.458,396.931,-103.642,176.468,30.090,155.268
C08652=1079.464,397.177,-103.682,176.472,30.098,155.270
C08653=1079.471,397.424,-103.722,176.476,30.106,155.271
C08654=1079.478,397.670,-103.762,176.480,30.114,155.273
C08655=1079.485,397.917,-103.802,176.484,30.123,155.275
C08656=1079.491,398.157,-103.842,176.489,30.131,155.276
C08657=1079.498,398.397,-103.881,176.492,30.139,155.278
C08658=1079.505,398.638,-103.920,176.496,30.147,155.280
C08659=1079.510,398.878,-103.959,176.500,30.155,155.281
C08660=1079.517,399.118,-103.999,176.504,30.163,155.283
C08661=1079.524,399.359,-104.038,176.509,30.171,155.285
C08662=1079.531,399.598,-104.078,176.512,30.179,155.286
C08663=1079.536,399.839,-104.117,176.516,30.188,155.288
C08664=1079.543,400.086,-104.158,176.520,30.196,155.290
C08665=1079.550,400.332,-104.198,176.524,30.204,155.292
C08666=1079.556,400.578,-104.239,176.528,30.213,155.293
C08667=1079.563,400.826,-104.279,176.533,30.222,155.295
C08668=1079.570,401.071,-104.320,176.537,30.230,155.297
C08669=1079.577,401.319,-104.360,176.541,30.238,155.299
C08670=1079.583,401.565,-104.401,176.545,30.247,155.300
C08671=1079.591,401.812,-104.442,176.549,30.256,155.302
C08672=1079.597,402.058,-104.482,176.554,30.264,155.304
C08673=1079.604,402.305,-104.523,176.558,30.273,155.306
C08674=1079.610,402.552,-104.564,176.562,30.282,155.308
C08675=1079.617,402.798,-104.605,176.566,30.290,155.309
C08676=1079.624,403.044,-104.646,176.570,30.299,155.311
C08677=1079.631,403.291,-104.687,176.574,30.308,155.313
C08678=1079.638,403.537,-104.727,176.579,30.316,155.315
C08679=1079.645,403.785,-104.768,176.583,30.325,155.317
C08680=1079.651,404.030,-104.809,176.587,30.334,155.319
C08681=1079.658,404.277,-104.851,176.591,30.343,155.320
C08682=1079.664,404.524,-104.891,176.595,30.351,155.322
C08683=1079.672,404.770,-104.932,176.599,30.360,155.324
C08684=1079.679,405.017,-104.973,176.604,30.369,155.326
C08685=1079.685,405.263,-105.015,176.608,30.378,155.328
C08686=1079.692,405.510,-105.056,176.612,30.387,155.330
C08687=1079.699,405.756,-105.097,176.616,30.396,155.332
C08688=1079.705,406.003,-105.138,176.621,30.405,155.334
C08689=1079.712,406.250,-105.179,176.626,30.414,155.336
C08690=1079.719,406.496,-105.220,176.630,30.424,155.337
C08691=1079.725,406.743,-105.262,176.634,30.433,155.339
C08692=1079.732,406.989,-105.303,176.638,30.442,155.341
C08693=1079.739,407.235,-105.344,176.642,30.451,155.343
C08694=1079.746,407.482,-105.386,176.647,30.460,155.345
C08695=1079.753,407.728,-105.427,176.651,30.469,155.347
C08696=1079.759,407.975,-105.468,176.656,30.478,155.349
C08697=1079.767,408.221,-105.510,176.660,30.487,155.351
C08698=1079.773,408.468,-105.552,176.664,30.497,155.353
C08699=1079.780,408.714,-105.593,176.668,30.506,155.355
C08700=1079.787,408.961,-105.635,176.673,30.516,155.357
C08701=1079.794,409.207,-105.676,176.677,30.525,155.359
C08702=1079.800,409.453,-105.718,176.682,30.534,155.361
C08703=1079.807,409.700,-105.760,176.686,30.544,155.363
C08704=1079.814,409.946,-105.801,176.690,30.553,155.365
C08705=1079.821,410.193,-105.844,176.695,30.562,155.367
C08706=1079.828,410.439,-105.885,176.700,30.572,155.369
C08707=1079.834,410.685,-105.927,176.704,30.582,155.371
C08708=1079.842,410.931,-105.968,176.708,30.591,155.373
C08709=1079.848,411.178,-106.010,176.712,30.601,155.375
C08710=1079.855,411.425,-106.053,176.718,30.610,155.377
C08711=1079.862,411.671,-106.094,176.722,30.620,155.379
C08712=1079.869,411.913,-106.135,176.726,30.629,155.381
C08713=1079.876,412.154,-106.176,176.730,30.639,155.383
C08714=1079.883,412.395,-106.217,176.735,30.648,155.385
C08715=1079.889,412.637,-106.259,176.740,30.658,155.387
C08716=1079.896,412.878,-106.301,176.744,30.667,155.390
C08717=1079.903,413.119,-106.341,176.748,30.677,155.392
C08718=1079.910,413.361,-106.383,176.752,30.686,155.394
C08719=1079.917,413.602,-106.424,176.757,30.696,155.396
C08720=1079.924,413.848,-106.466,176.762,30.706,155.398
C08721=1079.931,414.095,-106.509,176.766,30.716,155.400
C08722=1079.938,414.341,-106.550,176.771,30.726,155.402
C08723=1079.945,414.587,-106.592,176.776,30.736,155.404
C08724=1079.952,414.834,-106.635,176.780,30.746,155.406
C08725=1079.959,415.080,-106.677,176.785,30.755,155.408
C08726=1079.966,415.326,-106.719,176.789,30.765,155.411
C08727=1079.973,415.572,-106.762,176.794,30.775,155.413
C08728=1079.981,415.819,-106.805,176.799,30.785,155.415
C08729=1079.988,416.065,-106.847,176.803,30.796,155.417
C08730=1079.995,416.312,-106.890,176.808,30.806,155.419
C08731=1080.001,416.558,-106.932,176.812,30.816,155.422
C08732=1080.008,416.804,-106.975,176.818,30.827,155.424
C08733=1080.015,417.051,-107.018,176.822,30.836,155.426
C08734=1080.022,417.297,-107.060,176.827,30.847,155.428
C08735=1080.029,417.543,-107.103,176.831,30.858,155.431
C08736=1080.036,417.789,-107.146,176.837,30.868,155.433
C08737=1080.043,418.035,-107.188,176.841,30.878,155.435
C08738=1080.050,418.281,-107.231,176.846,30.889,155.438
C08739=1080.057,418.528,-107.275,176.850,30.899,155.440
C08740=1080.064,418.774,-107.317,176.856,30.909,155.442
C08741=1080.071,419.020,-107.360,176.860,30.920,155.444
C08742=1080.078,419.266,-107.403,176.865,30.930,155.447
C08743=1080.085,419.512,-107.445,176.869,30.941,155.449
C08744=1080.093,419.759,-107.489,176.875,30.952,155.451
C08745=1080.100,420.005,-107.532,176.879,30.962,155.454
C08746=1080.107,420.251,-107.575,176.884,30.973,155.456
C08747=1080.114,420.497,-107.617,176.889,30.984,155.458
C08748=1080.122,420.743,-107.661,176.894,30.994,155.461
C08749=1080.129,420.989,-107.704,176.899,31.005,155.463
C08750=1080.136,421.235,-107.747,176.903,31.016,155.465
C08751=1080.143,421.482,-107.790,176.908,31.027,155.468
C08752=1080.150,421.727,-107.834,176.914,31.037,155.470
C08753=1080.157,421.974,-107.876,176.918,31.048,155.473
C08754=1080.164,422.220,-107.920,176.923,31.059,155.475
C08755=1080.172,422.466,-107.964,176.928,31.070,155.477
C08756=1080.179,422.712,-108.007,176.933,31.081,155.480
C08757=1080.186,422.958,-108.051,176.938,31.092,155.482
C08758=1080.193,423.204,-108.094,176.942,31.103,155.485
C08759=1080.201,423.450,-108.138,176.948,31.115,155.487
C08760=1080.208,423.696,-108.181,176.953,31.126,155.490
C08761=1080.214,423.942,-108.225,176.958,31.137,155.492
C08762=1080.222,424.188,-108.269,176.963,31.148,155.495
C08763=1080.229,424.434,-108.312,176.968,31.159,155.497
C08764=1080.236,424.681,-108.356,176.973,31.171,155.500
C08765=1080.243,424.926,-108.400,176.978,31.182,155.502
C08766=1080.250,425.173,-108.444,176.983,31.193,155.505
C08767=1080.258,425.419,-108.487,176.988,31.205,155.507
C08768=1080.266,425.680,-108.534,176.993,31.217,155.510
C08769=1080.273,425.941,-108.580,176.999,31.229,155.513
C08770=1080.281,426.202,-108.627,177.004,31.241,155.515
C08771=1080.288,426.463,-108.674,177.010,31.253,155.518
C08772=1080.296,426.709,-108.717,177.015,31.265,155.521
C08773=1080.304,426.954,-108.761,177.020,31.277,155.523
C08774=1080.311,427.201,-108.806,177.025,31.288,155.526
C08775=1080.319,427.446,-108.850,177.031,31.300,155.529
C08776=1080.325,427.692,-108.894,177.036,31.312,155.531
C08777=1080.333,427.938,-108.938,177.041,31.323,155.534
C08778=1080.340,428.185,-108.982,177.047,31.335,155.537
C08779=1080.348,428.430,-109.026,177.051,31.347,155.539
C08780=1080.355,428.677,-109.071,177.056,31.359,155.542
C08781=1080.362,428.923,-109.115,177.062,31.371,155.545
C08782=1080.369,429.168,-109.159,177.067,31.383,155.547
C08783=1080.377,429.414,-109.204,177.072,31.395,155.550
C08784=1080.384,429.660,-109.249,177.078,31.407,155.553
C08785=1080.391,429.905,-109.293,177.083,31.419,155.555
C08786=1080.399,430.151,-109.337,177.089,31.431,155.558
C08787=1080.406,430.398,-109.382,177.094,31.443,155.561
C08788=1080.414,430.643,-109.427,177.099,31.455,155.564
C08789=1080.421,430.889,-109.471,177.105,31.467,155.566
C08790=1080.428,431.135,-109.516,177.110,31.480,155.569
C08791=1080.436,431.380,-109.561,177.115,31.492,155.572
C08792=1080.443,431.626,-109.605,177.121,31.505,155.575
C08793=1080.451,431.873,-109.650,177.126,31.517,155.578
C08794=1080.459,432.118,-109.695,177.132,31.529,155.581
C08795=1080.466,432.364,-109.740,177.137,31.542,155.583
C08796=1080.473,432.610,-109.784,177.143,31.554,155.586
C08797=1080.481,432.855,-109.830,177.148,31.567,155.589
C08798=1080.488,433.101,-109.875,177.153,31.579,155.592
C08799=1080.495,433.347,-109.920,177.159,31.592,155.595
C08800=1080.503,433.593,-109.965,177.164,31.605,155.598
C08801=1080.510,433.839,-110.010,177.170,31.618,155.601
C08802=1080.518,434.085,-110.055,177.175,31.630,155.604
C08803=1080.525,434.330,-110.101,177.181,31.643,155.606
C08804=1080.532,434.576,-110.145,177.187,31.656,155.609
C08805=1080.540,434.821,-110.191,177.192,31.669,155.612
C08806=1080.547,435.067,-110.236,177.198,31.682,155.615
C08807=1080.555,435.312,-110.282,177.203,31.695,155.618
C08808=1080.562,435.558,-110.327,177.209,31.708,155.621
C08809=1080.569,435.804,-110.372,177.214,31.721,155.624
C08810=1080.577,436.049,-110.418,177.221,31.734,155.627
C08811=1080.585,436.296,-110.464,177.226,31.747,155.630
C08812=1080.592,436.537,-110.508,177.232,31.760,155.633
C08813=1080.600,436.778,-110.552,177.237,31.773,155.636
C08814=1080.608,437.020,-110.598,177.243,31.786,155.639
C08815=1080.616,437.263,-110.642,177.248,31.799,155.642
C08816=1080.623,437.504,-110.688,177.255,31.813,155.646
C08817=1080.631,437.746,-110.732,177.260,31.826,155.649
C08818=1080.638,437.988,-110.778,177.266,31.839,155.652
C08819=1080.645,438.229,-110.823,177.271,31.852,155.655
C08820=1080.653,438.475,-110.869,177.277,31.866,155.658
C08821=1080.661,438.721,-110.915,177.284,31.879,155.661
C08822=1080.669,438.966,-110.961,177.289,31.893,155.664
C08823=1080.676,439.212,-111.006,177.295,31.907,155.667
C08824=1080.684,439.444,-111.050,177.300,31.920,155.670
C08825=1080.691,439.677,-111.093,177.306,31.933,155.673
C08826=1080.699,439.909,-111.137,177.312,31.946,155.676
C08827=1080.706,440.142,-111.181,177.318,31.959,155.680
C08828=1080.713,440.375,-111.225,177.324,31.972,155.683
C08829=1080.720,440.608,-111.268,177.329,31.985,155.686
C08830=1080.728,440.840,-111.312,177.335,31.999,155.689
C08831=1080.735,441.072,-111.356,177.340,32.012,155.692
C08832=1080.742,441.318,-111.402,177.346,32.026,155.695
C08833=1080.751,441.564,-111.449,177.353,32.041,155.699
C08834=1080.759,441.809,-111.495,177.358,32.054,155.702
C08835=1080.766,442.055,-111.542,177.365,32.069,155.705
C08836=1080.774,442.300,-111.588,177.371,32.083,155.709
C08837=1080.781,442.545,-111.635,177.377,32.098,155.712
C08838=1080.790,442.791,-111.681,177.383,32.112,155.715
C08839=1080.797,443.036,-111.728,177.389,32.127,155.719
C08840=1080.806,443.282,-111.775,177.395,32.141,155.722
C08841=1080.813,443.527,-111.822,177.402,32.156,155.726
C08842=1080.821,443.772,-111.869,177.408,32.170,155.729
C08843=1080.828,444.018,-111.915,177.414,32.185,155.732
C08844=1080.837,444.263,-111.962,177.421,32.199,155.736
C08845=1080.844,444.509,-112.009,177.427,32.214,155.739
C08846=1080.853,444.753,-112.056,177.433,32.229,155.743
C08847=1080.861,444.999,-112.103,177.439,32.244,155.747
C08848=1080.869,445.244,-112.150,177.446,32.259,155.750
C08849=1080.876,445.490,-112.197,177.452,32.274,155.754
C08850=1080.884,445.735,-112.244,177.458,32.289,155.757
C08851=1080.892,445.981,-112.291,177.465,32.304,155.761
C08852=1080.900,446.226,-112.339,177.471,32.319,155.764
C08853=1080.907,446.471,-112.386,177.477,32.334,155.768
C08854=1080.916,446.716,-112.433,177.482,32.349,155.772
C08855=1080.924,446.962,-112.481,177.487,32.364,155.775
C08856=1080.932,447.207,-112.528,177.492,32.379,155.779
C08857=1080.940,447.452,-112.575,177.497,32.394,155.783
C08858=1080.948,447.697,-112.622,177.502,32.409,155.786
C08859=1080.956,447.943,-112.670,177.506,32.424,155.790
C08860=1080.964,448.188,-112.718,177.510,32.440,155.794
C08861=1080.973,448.433,-112.765,177.514,32.454,155.797
C08862=1080.980,448.678,-112.813,177.518,32.469,155.801
C08863=1080.988,448.924,-112.860,177.521,32.484,155.805
C08864=1080.997,449.167,-112.908,177.525,32.499,155.808
C08865=1081.006,449.413,-112.954,177.528,32.513,155.812
C08866=1081.017,449.659,-113.000,177.531,32.527,155.815
C08867=1081.031,449.905,-113.045,177.534,32.539,155.818
C08868=1080.664,449.898,-113.265,177.507,32.709,155.864
C08869=1080.651,449.651,-113.221,177.504,32.696,155.860
C08870=1080.640,449.406,-113.175,177.500,32.683,155.857
C08871=1080.630,449.160,-113.128,177.497,32.669,155.853
C08872=1080.621,448.917,-113.080,177.493,32.654,155.850
C08873=1080.613,448.671,-113.033,177.490,32.639,155.846
C08874=1080.605,448.426,-112.985,177.486,32.624,155.842
C08875=1080.596,448.181,-112.938,177.482,32.609,155.839
C08876=1080.589,447.936,-112.891,177.477,32.594,155.835
C08877=1080.581,447.690,-112.843,177.474,32.579,155.831
C08878=1080.572,447.446,-112.795,177.469,32.564,155.828
C08879=1080.564,447.200,-112.748,177.464,32.549,155.824
C08880=1080.556,446.955,-112.700,177.459,32.534,155.820
C08881=1080.549,446.709,-112.653,177.453,32.519,155.817
C08882=1080.540,446.465,-112.605,177.447,32.503,155.813
C08883=1080.532,446.219,-112.558,177.441,32.488,155.809
C08884=1080.524,445.974,-112.510,177.435,32.473,155.806
C08885=1080.516,445.729,-112.464,177.429,32.458,155.802
C08886=1080.509,445.483,-112.416,177.422,32.443,155.799
C08887=1080.500,445.238,-112.368,177.416,32.428,155.795
C08888=1080.492,444.993,-112.322,177.410,32.414,155.792
C08889=1080.485,444.747,-112.275,177.403,32.398,155.788
C08890=1080.476,444.502,-112.228,177.396,32.384,155.784
C08891=1080.469,444.256,-112.181,177.390,32.369,155.781
C08892=1080.460,444.011,-112.134,177.384,32.354,155.777
C08893=1080.453,443.766,-112.087,177.378,32.340,155.774
C08894=1080.445,443.520,-112.040,177.371,32.325,155.770
C08895=1080.437,443.275,-111.993,177.364,32.310,155.767
C08896=1080.429,443.030,-111.947,177.359,32.296,155.764
C08897=1080.422,442.785,-111.900,177.352,32.281,155.760
C08898=1080.413,442.539,-111.853,177.346,32.267,155.757
C08899=1080.406,442.294,-111.806,177.339,32.252,155.753
C08900=1080.398,442.048,-111.760,177.334,32.238,155.750
C08901=1080.390,441.803,-111.713,177.327,32.224,155.747
C08902=1080.382,441.557,-111.666,177.321,32.210,155.743
C08903=1080.374,441.312,-111.621,177.315,32.196,155.740
C08904=1080.367,441.067,-111.574,177.309,32.181,155.737
C08905=1080.359,440.842,-111.532,177.303,32.168,155.734
C08906=1080.352,440.617,-111.489,177.297,32.156,155.731
C08907=1080.345,440.393,-111.447,177.292,32.143,155.728
C08908=1080.338,440.168,-111.405,177.287,32.130,155.725
C08909=1080.331,439.944,-111.362,177.281,32.118,155.722
C08910=1080.323,439.720,-111.320,177.275,32.105,155.719
C08911=1080.317,439.495,-111.278,177.270,32.092,155.716
C08912=1080.310,439.271,-111.235,177.264,32.079,155.713
C08913=1080.302,439.025,-111.189,177.258,32.066,155.710
C08914=1080.294,438.780,-111.144,177.253,32.052,155.707
C08915=1080.287,438.534,-111.098,177.246,32.038,155.703
C08916=1080.278,438.288,-111.052,177.241,32.025,155.700
C08917=1080.271,438.043,-111.007,177.235,32.011,155.697
C08918=1080.263,437.798,-110.960,177.228,31.998,155.694
C08919=1080.255,437.552,-110.915,177.223,31.985,155.691
C08920=1080.248,437.307,-110.868,177.217,31.971,155.688
C08921=1080.240,437.061,-110.822,177.211,31.958,155.685
C08922=1080.233,436.815,-110.777,177.205,31.945,155.682
C08923=1080.225,436.569,-110.732,177.199,31.931,155.678
C08924=1080.217,436.324,-110.686,177.194,31.918,155.675
C08925=1080.210,436.078,-110.640,177.188,31.905,155.672
C08926=1080.202,435.833,-110.595,177.183,31.892,155.669
C08927=1080.194,435.587,-110.549,177.176,31.879,155.666
C08928=1080.187,435.341,-110.504,177.170,31.866,155.663
C08929=1080.180,435.096,-110.459,177.165,31.853,155.660
C08930=1080.172,434.850,-110.413,177.159,31.840,155.657
C08931=1080.165,434.604,-110.368,177.154,31.827,155.654
C08932=1080.157,434.359,-110.322,177.148,31.814,155.651
C08933=1080.150,434.113,-110.277,177.143,31.801,155.648
C08934=1080.142,433.867,-110.232,177.137,31.788,155.646
C08935=1080.135,433.621,-110.187,177.131,31.775,155.643
C08936=1080.126,433.376,-110.142,177.125,31.763,155.640
C08937=1080.119,433.130,-110.097,177.120,31.750,155.637
C08938=1080.112,432.884,-110.052,177.114,31.737,155.634
C08939=1080.104,432.639,-110.006,177.109,31.725,155.631
C08940=1080.097,432.393,-109.961,177.103,31.713,155.628
C08941=1080.089,432.147,-109.916,177.098,31.700,155.625
C08942=1080.082,431.901,-109.871,177.092,31.687,155.622
C08943=1080.074,431.656,-109.827,177.087,31.675,155.620
C08944=1080.067,431.410,-109.782,177.081,31.663,155.617
C08945=1080.059,431.164,-109.737,177.076,31.651,155.614
C08946=1080.052,430.918,-109.692,177.070,31.638,155.611
C08947=1080.044,430.672,-109.648,177.065,31.626,155.608
C08948=1080.037,430.426,-109.603,177.059,31.614,155.606
C08949=1080.030,430.181,-109.558,177.054,31.601,155.603
C08950=1080.022,429.935,-109.514,177.048,31.590,155.600
C08951=1080.015,429.688,-109.470,177.043,31.578,155.597
C08952=1080.008,429.442,-109.425,177.038,31.565,155.595
C08953=1080.000,429.197,-109.381,177.032,31.553,155.592
C08954=1079.993,428.951,-109.336,177.028,31.541,155.589
C08955=1079.985,428.705,-109.291,177.022,31.529,155.587
C08956=1079.978,428.460,-109.248,177.017,31.518,155.584
C08957=1079.971,428.213,-109.203,177.011,31.506,155.581
C08958=1079.963,427.968,-109.158,177.006,31.494,155.578
C08959=1079.956,427.721,-109.114,177.000,31.482,155.576
C08960=1079.948,427.476,-109.070,176.995,31.470,155.573
C08961=1079.941,427.229,-109.026,176.991,31.459,155.571
C08962=1079.933,426.984,-108.982,176.985,31.447,155.568
C08963=1079.927,426.738,-108.938,176.980,31.435,155.565
C08964=1079.919,426.492,-108.893,176.974,31.424,155.563
C08965=1079.912,426.237,-108.848,176.969,31.412,155.560
C08966=1079.904,425.982,-108.802,176.964,31.400,155.557
C08967=1079.896,425.727,-108.757,176.958,31.388,155.555
C08968=1079.889,425.473,-108.711,176.953,31.376,155.552
C08969=1079.881,425.226,-108.668,176.948,31.365,155.550
C08970=1079.875,424.980,-108.624,176.943,31.354,155.547
C08971=1079.867,424.734,-108.580,176.938,31.342,155.544
C08972=1079.860,424.489,-108.536,176.932,31.331,155.542
C08973=1079.852,424.233,-108.491,176.927,31.319,155.539
C08974=1079.844,423.978,-108.445,176.922,31.308,155.537
C08975=1079.838,423.722,-108.400,176.916,31.296,155.534
C08976=1079.830,423.466,-108.355,176.911,31.285,155.532
C08977=1079.823,423.221,-108.312,176.907,31.273,155.529
C08978=1079.815,422.974,-108.268,176.901,31.262,155.527
C08979=1079.809,422.728,-108.224,176.896,31.251,155.524
C08980=1079.801,422.482,-108.181,176.892,31.240,155.522
C08981=1079.794,422.236,-108.137,176.886,31.229,155.519
C08982=1079.787,421.990,-108.093,176.882,31.218,155.517
C08983=1079.780,421.744,-108.050,176.876,31.207,155.514
C08984=1079.772,421.498,-108.007,176.871,31.196,155.512
C08985=1079.766,421.252,-107.964,176.867,31.185,155.510
C08986=1079.758,421.006,-107.920,176.861,31.175,155.507
C08987=1079.751,420.760,-107.877,176.856,31.164,155.505
C08988=1079.744,420.514,-107.835,176.852,31.153,155.503
C08989=1079.736,420.267,-107.791,176.846,31.142,155.500
C08990=1079.729,420.022,-107.748,176.842,31.132,155.498
C08991=1079.722,419.775,-107.705,176.837,31.121,155.496
C08992=1079.714,419.529,-107.662,176.832,31.111,155.493
C08993=1079.707,419.283,-107.619,176.827,31.100,155.491
C08994=1079.700,419.037,-107.576,176.823,31.089,155.488
C08995=1079.693,418.791,-107.533,176.818,31.079,155.486
C08996=1079.686,418.544,-107.490,176.813,31.069,155.484
C08997=1079.679,418.298,-107.447,176.808,31.058,155.482
C08998=1079.672,418.052,-107.405,176.804,31.048,155.479
C08999=1079.665,417.806,-107.361,176.798,31.037,155.477
C09000=1079.658,417.560,-107.319,176.794,31.027,155.475
C09001=1079.651,417.314,-107.276,176.789,31.017,155.473
C09002=1079.644,417.067,-107.233,176.784,31.006,155.470
C09003=1079.636,416.821,-107.190,176.779,30.996,155.468
C09004=1079.630,416.575,-107.148,176.775,30.986,155.466
C09005=1079.623,416.328,-107.105,176.769,30.976,155.464
C09006=1079.616,416.082,-107.062,176.765,30.965,155.461
C09007=1079.609,415.836,-107.020,176.761,30.955,155.459
C09008=1079.602,415.590,-106.977,176.756,30.945,155.457
C09009=1079.595,415.343,-106.935,176.751,30.935,155.455
C09010=1079.588,415.097,-106.892,176.746,30.925,155.453
C09011=1079.580,414.850,-106.850,176.742,30.915,155.450
C09012=1079.573,414.604,-106.807,176.737,30.905,155.448
C09013=1079.567,414.358,-106.765,176.732,30.895,155.446
C09014=1079.559,414.112,-106.723,176.728,30.885,155.444
C09015=1079.552,413.866,-106.680,176.723,30.875,155.442
C09016=1079.546,413.619,-106.639,176.718,30.865,155.440
C09017=1079.538,413.382,-106.597,176.714,30.856,155.438
C09018=1079.532,413.144,-106.557,176.710,30.846,155.436
C09019=1079.525,412.907,-106.517,176.705,30.837,155.434
C09020=1079.518,412.670,-106.476,176.701,30.828,155.432
C09021=1079.512,412.432,-106.436,176.697,30.819,155.430
C09022=1079.505,412.195,-106.396,176.691,30.809,155.427
C09023=1079.498,411.957,-106.355,176.687,30.800,155.426
C09024=1079.491,411.720,-106.315,176.683,30.790,155.424
C09025=1079.484,411.473,-106.272,176.679,30.781,155.421
C09026=1079.477,411.227,-106.230,176.674,30.771,155.419
C09027=1079.471,410.981,-106.189,176.669,30.762,155.417
C09028=1079.464,410.735,-106.146,176.665,30.752,155.415
C09029=1079.457,410.488,-106.105,176.660,30.743,155.413
C09030=1079.450,410.241,-106.063,176.656,30.733,155.411
C09031=1079.442,409.995,-106.021,176.652,30.724,155.409
C09032=1079.436,409.749,-105.979,176.647,30.714,155.407
C09033=1079.430,409.503,-105.937,176.642,30.705,155.405
C09034=1079.422,409.256,-105.896,176.638,30.696,155.403
C09035=1079.416,409.009,-105.854,176.634,30.686,155.401
C09036=1079.408,408.763,-105.813,176.630,30.677,155.399
C09037=1079.402,408.517,-105.771,176.624,30.667,155.397
C09038=1079.395,408.271,-105.729,176.620,30.658,155.395
C09039=1079.388,408.024,-105.688,176.616,30.649,155.393
C09040=1079.381,407.777,-105.646,176.612,30.639,155.391
C09041=1079.375,407.531,-105.605,176.607,30.630,155.389
C09042=1079.368,407.285,-105.563,176.603,30.621,155.387
C09043=1079.361,407.038,-105.521,176.599,30.612,155.385
C09044=1079.354,406.792,-105.480,176.595,30.603,155.383
C09045=1079.347,406.546,-105.439,176.590,30.593,155.381
C09046=1079.340,406.299,-105.397,176.585,30.584,155.379
C09047=1079.334,406.053,-105.356,176.581,30.575,155.378
C09048=1079.327,405.806,-105.315,176.577,30.566,155.376
C09049=1079.320,405.559,-105.274,176.573,30.557,155.374
C09050=1079.314,405.313,-105.233,176.568,30.549,155.372
C09051=1079.306,405.066,-105.192,176.564,30.540,155.370
C09052=1079.300,404.820,-105.150,176.560,30.531,155.368
C09053=1079.293,404.573,-105.109,176.556,30.522,155.366
C09054=1079.286,404.327,-105.068,176.551,30.513,155.364
C09055=1079.279,404.080,-105.028,176.547,30.504,155.362
C09056=1079.273,403.833,-104.986,176.543,30.495,155.361
C09057=1079.266,403.588,-104.945,176.539,30.486,155.359
C09058=1079.259,403.340,-104.905,176.534,30.478,155.357
C09059=1079.252,403.094,-104.864,176.530,30.469,155.355
C09060=1079.245,402.848,-104.823,176.526,30.460,155.353
C09061=1079.238,402.601,-104.782,176.522,30.452,155.351
C09062=1079.232,402.355,-104.741,176.517,30.443,155.350
C09063=1079.225,402.107,-104.700,176.513,30.434,155.348
C09064=1079.219,401.861,-104.659,176.509,30.426,155.346
C09065=1079.212,401.614,-104.619,176.505,30.417,155.344
C09066=1079.205,401.368,-104.578,176.501,30.409,155.342
C09067=1079.199,401.122,-104.538,176.496,30.400,155.341
C09068=1079.191,400.875,-104.496,176.492,30.392,155.339
C09069=1079.185,400.629,-104.456,176.488,30.383,155.337
C09070=1079.178,400.382,-104.415,176.484,30.374,155.335
C09071=1079.171,400.135,-104.375,176.479,30.366,155.334
C09072=1079.165,399.889,-104.335,176.475,30.357,155.332
C09073=1079.158,399.648,-104.295,176.471,30.349,155.330
C09074=1079.152,399.407,-104.255,176.468,30.341,155.328
C09075=1079.145,399.166,-104.216,176.463,30.333,155.327
C09076=1079.138,398.925,-104.176,176.459,30.325,155.325
C09077=1079.132,398.684,-104.137,176.455,30.317,155.323
C09078=1079.125,398.443,-104.097,176.451,30.308,155.322
C09079=1079.118,398.202,-104.058,176.448,30.301,155.320
C09080=1079.112,397.961,-104.018,176.443,30.292,155.318
C09081=1079.106,397.714,-103.978,176.439,30.284,155.317
C09082=1079.098,397.468,-103.938,176.435,30.276,155.315
C09083=1079.092,397.222,-103.898,176.431,30.268,155.313
C09084=1079.085,396.975,-103.858,176.426,30.259,155.311
C09085=1079.079,396.728,-103.818,176.423,30.252,155.310
C09086=1079.072,396.482,-103.778,176.419,30.243,155.308
